LIN {X 0,Y 164.353,Z 359.01,A -85,B 0,C 180,E1 -23368.785,E2 -23368.785} C_VEL
LIN {X 0,Y 164.395,Z 359.001,A -85,B 0,C 180,E1 -23374.69,E2 -23374.69} C_VEL
LIN {X 0,Y 164.485,Z 358.995,A -85,B 0,C 180,E1 -23380.051,E2 -23380.051} C_VEL
LIN {X 0,Y 164.525,Z 358.989,A -85,B 0,C 180,E1 -23385.149,E2 -23385.149} C_VEL
LIN {X 0,Y 164.803,Z 358.955,A -85,B 0,C 180,E1 -23390.178,E2 -23390.178} C_VEL
LIN {X 0,Y 164.851,Z 358.949,A -85,B 0,C 180,E1 -23392.652,E2 -23392.652} C_VEL
LIN {X 0,Y 165.049,Z 358.926,A -85,B 0,C 180,E1 -23397.559,E2 -23397.559} C_VEL
LIN {X 0,Y 165.289,Z 358.897,A -85,B 0,C 180,E1 -23400,E2 -23400} C_VEL
LIN {X 0,Y 164.763,Z 358.963,A -85,B 0,C 180,E1 -23404.894,E2 -23404.894} C_VEL
LIN {X 0,Y 164.831,Z 358.955,A -85,B 0,C 180,E1 -23407.349,E2 -23407.349} C_VEL
LIN {X 0,Y 164.703,Z 358.969,A -85,B 0,C 180,E1 -23411.061,E2 -23411.061} C_VEL
LIN {X 0,Y 164.483,Z 358.999,A -85,B 0,C 180,E1 -23417.403,E2 -23417.403} C_VEL
LIN {X 0,Y 164.474,Z 358.998,A -85,B 0,C 180,E1 -23419.989,E2 -23419.989} C_VEL
LIN {X 0,Y 164.395,Z 359.008,A -85,B 0,C 180,E1 -23425.309,E2 -23425.309} C_VEL
LIN {X 0,Y 164.82,Z 361.559,A -85,B 0,C 180,E1 -23431.481,E2 -23431.481} C_VEL
LIN {X 0,Y 165.147,Z 364.035,A -85,B 0,C 180,E1 -23436.569,E2 -23436.569} C_VEL
LIN {X 0,Y 165.54,Z 366.68,A -85,B 0,C 180,E1 -23441.479,E2 -23441.479} C_VEL
LIN {X 0,Y 166.739,Z 369.834,A -85,B 0,C 180,E1 -23442.221,E2 -23442.221} C_VEL
LIN {X 0,Y 168.781,Z 372.777,A -85,B 0,C 180,E1 -23443.252,E2 -23443.252} C_VEL
LIN {X 0,Y 170.799,Z 376.689,A -85,B 0,C 180,E1 -23444.388,E2 -23444.388} C_VEL
LIN {X 0,Y 174.052,Z 383.605,A -85,B 0,C 180,E1 -23446.305,E2 -23446.305} C_VEL
LIN {X 0,Y 176.79,Z 390.925,A -85,B 0,C 180,E1 -23448.191,E2 -23448.191} C_VEL
LIN {X 0,Y 178.354,Z 398.431,A -85,B 0,C 180,E1 -23449.912,E2 -23449.912} C_VEL
LIN {X 0,Y 179.413,Z 408.097,A -85,B 0,C 180,E1 -23452.121,E2 -23452.121} C_VEL
LIN {X 0,Y 179.618,Z 418.57,A -85,B 0,C 180,E1 -23454.683,E2 -23454.683} C_VEL
LIN {X 0,Y 178.968,Z 428.265,A -85,B 0,C 180,E1 -23457.319,E2 -23457.319} C_VEL
LIN {X 0,Y 178.405,Z 432.364,A -85,B 0,C 180,E1 -23458.535,E2 -23458.535} C_VEL
LIN {X 0,Y 175.059,Z 441.2,A -85,B 0,C 180,E1 -23461.199,E2 -23461.199} C_VEL
LIN {X 0,Y 172.159,Z 448.374,A -85,B 0,C 180,E1 -23463.91,E2 -23463.91} C_VEL
LIN {X 0,Y 168.88,Z 455.682,A -85,B 0,C 180,E1 -23467.359,E2 -23467.359} C_VEL
LIN {X 0,Y 166.696,Z 460.537,A -85,B 0,C 180,E1 -23470.288,E2 -23470.288} C_VEL
LIN {X 0,Y 164.537,Z 465.256,A -85,B 0,C 180,E1 -23473.88,E2 -23473.88} C_VEL
LIN {X 0,Y 163.144,Z 468.87,A -85,B 0,C 180,E1 -23477.561,E2 -23477.561} C_VEL
LIN {X 0,Y 162.461,Z 470.733,A -85,B 0,C 180,E1 -23480.035,E2 -23480.035} C_VEL
LIN {X 0,Y 161.852,Z 473.135,A -85,B 0,C 180,E1 -23485.017,E2 -23485.017} C_VEL
LIN {X 0,Y 161.797,Z 473.748,A -85,B 0,C 180,E1 -23487.509,E2 -23487.509} C_VEL
LIN {X 0,Y 161.893,Z 473.964,A -85,B 0,C 180,E1 -23489.999,E2 -23489.999} C_VEL
LIN {X 0,Y 161.797,Z 473.737,A -85,B 0,C 180,E1 -23492.488,E2 -23492.488} C_VEL
LIN {X 0,Y 161.851,Z 473.118,A -85,B 0,C 180,E1 -23494.981,E2 -23494.981} C_VEL
LIN {X 0,Y 162.035,Z 472.109,A -85,B 0,C 180,E1 -23497.475,E2 -23497.475} C_VEL
LIN {X 0,Y 162.46,Z 470.698,A -85,B 0,C 180,E1 -23499.963,E2 -23499.963} C_VEL
LIN {X 0,Y 163.562,Z 467.743,A -85,B 0,C 180,E1 -23503.668,E2 -23503.668} C_VEL
LIN {X 0,Y 165.152,Z 463.748,A -85,B 0,C 180,E1 -23507.329,E2 -23507.329} C_VEL
LIN {X 0,Y 167.969,Z 457.619,A -85,B 0,C 180,E1 -23511.474,E2 -23511.474} C_VEL
LIN {X 0,Y 170.947,Z 451.054,A -85,B 0,C 180,E1 -23514.857,E2 -23514.857} C_VEL
LIN {X 0,Y 173.3,Z 445.244,A -85,B 0,C 180,E1 -23517.303,E2 -23517.303} C_VEL
LIN {X 0,Y 174.216,Z 441.463,A -85,B 0,C 180,E1 -23518.769,E2 -23518.769} C_VEL
LIN {X 0,Y 174.238,Z 437.625,A -85,B 0,C 180,E1 -23520.281,E2 -23520.281} C_VEL
LIN {X 0,Y 173.009,Z 426.964,A -85,B 0,C 180,E1 -23524.249,E2 -23524.249} C_VEL
LIN {X 0,Y 173.036,Z 423.996,A -85,B 0,C 180,E1 -23525.153,E2 -23525.153} C_VEL
LIN {X 0,Y 173.396,Z 414.41,A -85,B 0,C 180,E1 -23527.76,E2 -23527.76} C_VEL
LIN {X 0,Y 172.882,Z 404.098,A -85,B 0,C 180,E1 -23530.339,E2 -23530.339} C_VEL
LIN {X 0,Y 171.558,Z 395.307,A -85,B 0,C 180,E1 -23532.491,E2 -23532.491} C_VEL
LIN {X 0,Y 169.041,Z 387.542,A -85,B 0,C 180,E1 -23534.604,E2 -23534.604} C_VEL
LIN {X 0,Y 165.953,Z 380.904,A -85,B 0,C 180,E1 -23536.66,E2 -23536.66} C_VEL
LIN {X 0,Y 163.83,Z 376.649,A -85,B 0,C 180,E1 -23538.014,E2 -23538.014} C_VEL
LIN {X 0,Y 161.813,Z 372.888,A -85,B 0,C 180,E1 -23539.276,E2 -23539.276} C_VEL
LIN {X 0,Y 160.79,Z 371.257,A -85,B 0,C 180,E1 -23539.868,E2 -23539.868} C_VEL
LIN {X 0,Y 158.767,Z 367.896,A -85,B 0,C 180,E1 -23541.098,E2 -23541.098} C_VEL
LIN {X 0,Y 158.284,Z 366.287,A -85,B 0,C 180,E1 -23541.566,E2 -23541.566} C_VEL
LIN {X 0,Y 158.063,Z 364.741,A -85,B 0,C 180,E1 -23544.688,E2 -23544.688} C_VEL
LIN {X 0,Y 157.879,Z 363.325,A -85,B 0,C 180,E1 -23547.752,E2 -23547.752} C_VEL
LIN {X 0,Y 157.498,Z 360.965,A -85,B 0,C 180,E1 -23553.498,E2 -23553.498} C_VEL
LIN {X 0,Y 157.295,Z 359.957,A -85,B 0,C 180,E1 -23556.289,E2 -23556.289} C_VEL
LIN {X 0,Y 157.405,Z 359.877,A -85,B 0,C 180,E1 -23561.787,E2 -23561.787} C_VEL
LIN {X 0,Y 157.542,Z 359.86,A -85,B 0,C 180,E1 -23567.112,E2 -23567.112} C_VEL
LIN {X 0,Y 157.741,Z 359.835,A -85,B 0,C 180,E1 -23569.734,E2 -23569.734} C_VEL
LIN {X 0,Y 157.807,Z 359.828,A -85,B 0,C 180,E1 -23572.322,E2 -23572.322} C_VEL
LIN {X 0,Y 158.246,Z 359.771,A -85,B 0,C 180,E1 -23580,E2 -23580} C_VEL
LIN {X 0,Y 157.815,Z 359.825,A -85,B 0,C 180,E1 -23587.678,E2 -23587.678} C_VEL
LIN {X 0,Y 157.672,Z 359.842,A -85,B 0,C 180,E1 -23591.311,E2 -23591.311} C_VEL
LIN {X 0,Y 157.449,Z 359.874,A -85,B 0,C 180,E1 -23595.535,E2 -23595.535} C_VEL
LIN {X 0,Y 157.362,Z 359.884,A -85,B 0,C 180,E1 -23600.934,E2 -23600.934} C_VEL
LIN {X 0,Y 157.305,Z 359.889,A -85,B 0,C 180,E1 -23606.682,E2 -23606.682} C_VEL
LIN {X 0,Y 157.263,Z 359.896,A -85,B 0,C 180,E1 -23612.431,E2 -23612.431} C_VEL
LIN {X 0,Y 157.275,Z 360.116,A -85,B 0,C 180,E1 -23616.456,E2 -23616.456} C_VEL
LIN {X 0,Y 157.298,Z 360.711,A -85,B 0,C 180,E1 -23618.163,E2 -23618.163} C_VEL
LIN {X 0,Y 158.359,Z 363.418,A -85,B 0,C 180,E1 -23618.941,E2 -23618.941} C_VEL
LIN {X 0,Y 160.846,Z 366.551,A -85,B 0,C 180,E1 -23620.375,E2 -23620.375} C_VEL
LIN {X 0,Y 162.74,Z 370.024,A -85,B 0,C 180,E1 -23621.604,E2 -23621.604} C_VEL
LIN {X 0,Y 163.87,Z 371.847,A -85,B 0,C 180,E1 -23622.284,E2 -23622.284} C_VEL
LIN {X 0,Y 166.98,Z 377.77,A -85,B 0,C 180,E1 -23624.318,E2 -23624.318} C_VEL
LIN {X 0,Y 170.348,Z 385.376,A -85,B 0,C 180,E1 -23626.767,E2 -23626.767} C_VEL
LIN {X 0,Y 172.965,Z 393.791,A -85,B 0,C 180,E1 -23629.227,E2 -23629.227} C_VEL
LIN {X 0,Y 174.476,Z 402.79,A -85,B 0,C 180,E1 -23631.718,E2 -23631.718} C_VEL
LIN {X 0,Y 175.187,Z 412.008,A -85,B 0,C 180,E1 -23634.384,E2 -23634.384} C_VEL
LIN {X 0,Y 175.109,Z 418.891,A -85,B 0,C 180,E1 -23636.507,E2 -23636.507} C_VEL
LIN {X 0,Y 171.621,Z 428.426,A -85,B 0,C 180,E1 -23639.195,E2 -23639.195} C_VEL
LIN {X 0,Y 168.381,Z 436.318,A -85,B 0,C 180,E1 -23641.996,E2 -23641.996} C_VEL
LIN {X 0,Y 164.694,Z 443.99,A -85,B 0,C 180,E1 -23645.416,E2 -23645.416} C_VEL
LIN {X 0,Y 161.143,Z 451.035,A -85,B 0,C 180,E1 -23649.581,E2 -23649.581} C_VEL
LIN {X 0,Y 158.778,Z 455.72,A -85,B 0,C 180,E1 -23653.281,E2 -23653.281} C_VEL
LIN {X 0,Y 157.001,Z 459.302,A -85,B 0,C 180,E1 -23657.068,E2 -23657.068} C_VEL
LIN {X 0,Y 156.157,Z 461.149,A -85,B 0,C 180,E1 -23659.63,E2 -23659.63} C_VEL
LIN {X 0,Y 155.58,Z 462.534,A -85,B 0,C 180,E1 -23662.213,E2 -23662.213} C_VEL
LIN {X 0,Y 154.905,Z 464.126,A -85,B 0,C 180,E1 -23667.401,E2 -23667.401} C_VEL
LIN {X 0,Y 154.879,Z 464.35,A -85,B 0,C 180,E1 -23670.001,E2 -23670.001} C_VEL
LIN {X 0,Y 154.976,Z 463.919,A -85,B 0,C 180,E1 -23673.9,E2 -23673.9} C_VEL
LIN {X 0,Y 155.515,Z 462.602,A -85,B 0,C 180,E1 -23677.793,E2 -23677.793} C_VEL
LIN {X 0,Y 156.164,Z 461.244,A -85,B 0,C 180,E1 -23680.372,E2 -23680.372} C_VEL
LIN {X 0,Y 157.501,Z 458.377,A -85,B 0,C 180,E1 -23684.208,E2 -23684.208} C_VEL
LIN {X 0,Y 159.461,Z 454.485,A -85,B 0,C 180,E1 -23687.97,E2 -23687.97} C_VEL
LIN {X 0,Y 161.987,Z 449.463,A -85,B 0,C 180,E1 -23691.641,E2 -23691.641} C_VEL
LIN {X 0,Y 165.187,Z 443.13,A -85,B 0,C 180,E1 -23695.18,E2 -23695.18} C_VEL
LIN {X 0,Y 168.859,Z 435.21,A -85,B 0,C 180,E1 -23698.597,E2 -23698.597} C_VEL
LIN {X 0,Y 172.096,Z 427.315,A -85,B 0,C 180,E1 -23701.31,E2 -23701.31} C_VEL
LIN {X 0,Y 175.172,Z 419.412,A -85,B 0,C 180,E1 -23703.481,E2 -23703.481} C_VEL
LIN {X 0,Y 175.141,Z 409.831,A -85,B 0,C 180,E1 -23706.414,E2 -23706.414} C_VEL
LIN {X 0,Y 174.237,Z 400.686,A -85,B 0,C 180,E1 -23709.03,E2 -23709.03} C_VEL
LIN {X 0,Y 172.483,Z 391.797,A -85,B 0,C 180,E1 -23711.52,E2 -23711.52} C_VEL
LIN {X 0,Y 169.319,Z 382.614,A -85,B 0,C 180,E1 -23714.274,E2 -23714.274} C_VEL
LIN {X 0,Y 165.221,Z 374.414,A -85,B 0,C 180,E1 -23717.034,E2 -23717.034} C_VEL
LIN {X 0,Y 162.756,Z 370.019,A -85,B 0,C 180,E1 -23718.607,E2 -23718.607} C_VEL
LIN {X 0,Y 160.857,Z 366.588,A -85,B 0,C 180,E1 -23719.839,E2 -23719.839} C_VEL
LIN {X 0,Y 157.969,Z 362.664,A -85,B 0,C 180,E1 -23721.554,E2 -23721.554} C_VEL
LIN {X 0,Y 157.322,Z 360.713,A -85,B 0,C 180,E1 -23722.081,E2 -23722.081} C_VEL
LIN {X 0,Y 157.278,Z 359.894,A -85,B 0,C 180,E1 -23724.485,E2 -23724.485} C_VEL
LIN {X 0,Y 157.28,Z 359.889,A -85,B 0,C 180,E1 -23728.104,E2 -23728.104} C_VEL
LIN {X 0,Y 157.31,Z 359.889,A -85,B 0,C 180,E1 -23733.464,E2 -23733.464} C_VEL
LIN {X 0,Y 157.393,Z 359.879,A -85,B 0,C 180,E1 -23739.67,E2 -23739.67} C_VEL
LIN {X 0,Y 157.455,Z 359.872,A -85,B 0,C 180,E1 -23744.466,E2 -23744.466} C_VEL
LIN {X 0,Y 157.727,Z 359.838,A -85,B 0,C 180,E1 -23749.733,E2 -23749.733} C_VEL
LIN {X 0,Y 157.808,Z 359.828,A -85,B 0,C 180,E1 -23752.322,E2 -23752.322} C_VEL
LIN {X 0,Y 158.252,Z 359.774,A -85,B 0,C 180,E1 -23760,E2 -23760} C_VEL
LIN {X 0,Y 157.768,Z 359.836,A -85,B 0,C 180,E1 -23767.68,E2 -23767.68} C_VEL
LIN {X 0,Y 157.638,Z 359.85,A -85,B 0,C 180,E1 -23771.236,E2 -23771.236} C_VEL
LIN {X 0,Y 157.453,Z 359.874,A -85,B 0,C 180,E1 -23775.534,E2 -23775.534} C_VEL
LIN {X 0,Y 157.368,Z 359.884,A -85,B 0,C 180,E1 -23780.933,E2 -23780.933} C_VEL
LIN {X 0,Y 157.309,Z 360.019,A -85,B 0,C 180,E1 -23783.709,E2 -23783.709} C_VEL
LIN {X 0,Y 157.506,Z 361.155,A -85,B 0,C 180,E1 -23786.822,E2 -23786.822} C_VEL
LIN {X 0,Y 157.912,Z 363.396,A -85,B 0,C 180,E1 -23792.281,E2 -23792.281} C_VEL
LIN {X 0,Y 158.272,Z 366.115,A -85,B 0,C 180,E1 -23797.974,E2 -23797.974} C_VEL
LIN {X 0,Y 158.312,Z 366.364,A -85,B 0,C 180,E1 -23798.426,E2 -23798.426} C_VEL
LIN {X 0,Y 159.319,Z 369.145,A -85,B 0,C 180,E1 -23799.151,E2 -23799.151} C_VEL
LIN {X 0,Y 161.764,Z 372.735,A -85,B 0,C 180,E1 -23800.567,E2 -23800.567} C_VEL
LIN {X 0,Y 163.614,Z 376.302,A -85,B 0,C 180,E1 -23801.744,E2 -23801.744} C_VEL
LIN {X 0,Y 164.947,Z 378.808,A -85,B 0,C 180,E1 -23802.563,E2 -23802.563} C_VEL
LIN {X 0,Y 168.731,Z 386.833,A -85,B 0,C 180,E1 -23805.079,E2 -23805.079} C_VEL
LIN {X 0,Y 171.42,Z 394.551,A -85,B 0,C 180,E1 -23807.241,E2 -23807.241} C_VEL
LIN {X 0,Y 172.895,Z 403.402,A -85,B 0,C 180,E1 -23809.429,E2 -23809.429} C_VEL
LIN {X 0,Y 173.449,Z 413.342,A -85,B 0,C 180,E1 -23811.9,E2 -23811.9} C_VEL
LIN {X 0,Y 173.197,Z 423.113,A -85,B 0,C 180,E1 -23814.541,E2 -23814.541} C_VEL
LIN {X 0,Y 172.16,Z 432.143,A -85,B 0,C 180,E1 -23817.255,E2 -23817.255} C_VEL
LIN {X 0,Y 170.986,Z 435.894,A -85,B 0,C 180,E1 -23818.394,E2 -23818.394} C_VEL
LIN {X 0,Y 167.504,Z 444.057,A -85,B 0,C 180,E1 -23821.15,E2 -23821.15} C_VEL
LIN {X 0,Y 163.992,Z 452.076,A -85,B 0,C 180,E1 -23824.623,E2 -23824.623} C_VEL
LIN {X 0,Y 160.925,Z 458.501,A -85,B 0,C 180,E1 -23828.209,E2 -23828.209} C_VEL
LIN {X 0,Y 158.373,Z 463.605,A -85,B 0,C 180,E1 -23831.902,E2 -23831.902} C_VEL
LIN {X 0,Y 156.631,Z 467.579,A -85,B 0,C 180,E1 -23835.712,E2 -23835.712} C_VEL
LIN {X 0,Y 155.458,Z 470.518,A -85,B 0,C 180,E1 -23839.581,E2 -23839.581} C_VEL
LIN {X 0,Y 154.757,Z 472.92,A -85,B 0,C 180,E1 -23844.788,E2 -23844.788} C_VEL
LIN {X 0,Y 154.712,Z 473.627,A -85,B 0,C 180,E1 -23847.982,E2 -23847.982} C_VEL
LIN {X 0,Y 154.794,Z 473.749,A -85,B 0,C 180,E1 -23849.999,E2 -23849.999} C_VEL
LIN {X 0,Y 154.699,Z 473.521,A -85,B 0,C 180,E1 -23852.603,E2 -23852.603} C_VEL
LIN {X 0,Y 154.757,Z 472.901,A -85,B 0,C 180,E1 -23855.21,E2 -23855.21} C_VEL
LIN {X 0,Y 154.98,Z 471.892,A -85,B 0,C 180,E1 -23857.818,E2 -23857.818} C_VEL
LIN {X 0,Y 155.456,Z 470.481,A -85,B 0,C 180,E1 -23860.417,E2 -23860.417} C_VEL
LIN {X 0,Y 156.63,Z 467.525,A -85,B 0,C 180,E1 -23864.286,E2 -23864.286} C_VEL
LIN {X 0,Y 158.371,Z 463.531,A -85,B 0,C 180,E1 -23868.096,E2 -23868.096} C_VEL
LIN {X 0,Y 161.322,Z 457.4,A -85,B 0,C 180,E1 -23872.406,E2 -23872.406} C_VEL
LIN {X 0,Y 164.722,Z 450.298,A -85,B 0,C 180,E1 -23876.158,E2 -23876.158} C_VEL
LIN {X 0,Y 168.114,Z 442.409,A -85,B 0,C 180,E1 -23879.418,E2 -23879.418} C_VEL
LIN {X 0,Y 171.641,Z 433.901,A -85,B 0,C 180,E1 -23882.159,E2 -23882.159} C_VEL
LIN {X 0,Y 172.781,Z 426.73,A -85,B 0,C 180,E1 -23884.357,E2 -23884.357} C_VEL
LIN {X 0,Y 173.036,Z 423.996,A -85,B 0,C 180,E1 -23885.153,E2 -23885.153} C_VEL
LIN {X 0,Y 172.687,Z 419.729,A -85,B 0,C 180,E1 -23886.491,E2 -23886.491} C_VEL
LIN {X 0,Y 171.451,Z 415.728,A -85,B 0,C 180,E1 -23887.905,E2 -23887.905} C_VEL
LIN {X 0,Y 168.105,Z 407.951,A -85,B 0,C 180,E1 -23890.782,E2 -23890.782} C_VEL
LIN {X 0,Y 166.636,Z 402.115,A -85,B 0,C 180,E1 -23892.582,E2 -23892.582} C_VEL
LIN {X 0,Y 165.321,Z 395.581,A -85,B 0,C 180,E1 -23894.395,E2 -23894.395} C_VEL
LIN {X 0,Y 163.025,Z 389.258,A -85,B 0,C 180,E1 -23896.389,E2 -23896.389} C_VEL
LIN {X 0,Y 159.585,Z 381.699,A -85,B 0,C 180,E1 -23898.969,E2 -23898.969} C_VEL
LIN {X 0,Y 156.809,Z 376.441,A -85,B 0,C 180,E1 -23900.93,E2 -23900.93} C_VEL
LIN {X 0,Y 154.709,Z 372.434,A -85,B 0,C 180,E1 -23902.445,E2 -23902.445} C_VEL
LIN {X 0,Y 151.861,Z 368.339,A -85,B 0,C 180,E1 -23904.35,E2 -23904.35} C_VEL
LIN {X 0,Y 151.071,Z 365.975,A -85,B 0,C 180,E1 -23905.055,E2 -23905.055} C_VEL
LIN {X 0,Y 150.802,Z 364.217,A -85,B 0,C 180,E1 -23909.16,E2 -23909.16} C_VEL
LIN {X 0,Y 150.593,Z 362.925,A -85,B 0,C 180,E1 -23912.458,E2 -23912.458} C_VEL
LIN {X 0,Y 150.279,Z 361,A -85,B 0,C 180,E1 -23918.029,E2 -23918.029} C_VEL
LIN {X 0,Y 150.354,Z 360.757,A -85,B 0,C 180,E1 -23920.901,E2 -23920.901} C_VEL
LIN {X 0,Y 150.445,Z 360.744,A -85,B 0,C 180,E1 -23926.493,E2 -23926.493} C_VEL
LIN {X 0,Y 150.658,Z 360.716,A -85,B 0,C 180,E1 -23929.246,E2 -23929.246} C_VEL
LIN {X 0,Y 150.744,Z 360.706,A -85,B 0,C 180,E1 -23931.96,E2 -23931.96} C_VEL
LIN {X 0,Y 151.208,Z 360.648,A -85,B 0,C 180,E1 -23940,E2 -23940} C_VEL
LIN {X 0,Y 150.75,Z 360.704,A -85,B 0,C 180,E1 -23948.04,E2 -23948.04} C_VEL
LIN {X 0,Y 150.608,Z 360.722,A -85,B 0,C 180,E1 -23951.505,E2 -23951.505} C_VEL
LIN {X 0,Y 150.356,Z 360.755,A -85,B 0,C 180,E1 -23956.287,E2 -23956.287} C_VEL
LIN {X 0,Y 150.345,Z 360.758,A -85,B 0,C 180,E1 -23960.791,E2 -23960.791} C_VEL
LIN {X 0,Y 150.234,Z 360.771,A -85,B 0,C 180,E1 -23967.279,E2 -23967.279} C_VEL
LIN {X 0,Y 150.204,Z 360.774,A -85,B 0,C 180,E1 -23972.629,E2 -23972.629} C_VEL
LIN {X 0,Y 150.223,Z 361.059,A -85,B 0,C 180,E1 -23974.559,E2 -23974.559} C_VEL
LIN {X 0,Y 151.303,Z 363.715,A -85,B 0,C 180,E1 -23975.495,E2 -23975.495} C_VEL
LIN {X 0,Y 153.858,Z 366.979,A -85,B 0,C 180,E1 -23977.218,E2 -23977.218} C_VEL
LIN {X 0,Y 155.877,Z 370.541,A -85,B 0,C 180,E1 -23978.703,E2 -23978.703} C_VEL
LIN {X 0,Y 157.095,Z 372.257,A -85,B 0,C 180,E1 -23979.502,E2 -23979.502} C_VEL
LIN {X 0,Y 161.032,Z 379.67,A -85,B 0,C 180,E1 -23982.399,E2 -23982.399} C_VEL
LIN {X 0,Y 164.489,Z 387.463,A -85,B 0,C 180,E1 -23985.171,E2 -23985.171} C_VEL
LIN {X 0,Y 166.872,Z 395.066,A -85,B 0,C 180,E1 -23987.637,E2 -23987.637} C_VEL
LIN {X 0,Y 168.396,Z 403.904,A -85,B 0,C 180,E1 -23990.304,E2 -23990.304} C_VEL
LIN {X 0,Y 169.005,Z 413.397,A -85,B 0,C 180,E1 -23993.234,E2 -23993.234} C_VEL
LIN {X 0,Y 168.812,Z 420.176,A -85,B 0,C 180,E1 -23995.444,E2 -23995.444} C_VEL
LIN {X 0,Y 165.544,Z 428.694,A -85,B 0,C 180,E1 -23997.952,E2 -23997.952} C_VEL
LIN {X 0,Y 162.145,Z 436.536,A -85,B 0,C 180,E1 -24000.818,E2 -24000.818} C_VEL
LIN {X 0,Y 158.275,Z 444.207,A -85,B 0,C 180,E1 -24004.348,E2 -24004.348} C_VEL
LIN {X 0,Y 154.492,Z 451.252,A -85,B 0,C 180,E1 -24008.66,E2 -24008.66} C_VEL
LIN {X 0,Y 151.996,Z 455.937,A -85,B 0,C 180,E1 -24012.511,E2 -24012.511} C_VEL
LIN {X 0,Y 150.075,Z 459.519,A -85,B 0,C 180,E1 -24016.46,E2 -24016.46} C_VEL
LIN {X 0,Y 149.17,Z 461.366,A -85,B 0,C 180,E1 -24019.139,E2 -24019.139} C_VEL
LIN {X 0,Y 148.544,Z 462.75,A -85,B 0,C 180,E1 -24021.841,E2 -24021.841} C_VEL
LIN {X 0,Y 147.825,Z 464.341,A -85,B 0,C 180,E1 -24027.276,E2 -24027.276} C_VEL
LIN {X 0,Y 147.782,Z 464.566,A -85,B 0,C 180,E1 -24030.001,E2 -24030.001} C_VEL
LIN {X 0,Y 147.84,Z 464.264,A -85,B 0,C 180,E1 -24033.339,E2 -24033.339} C_VEL
LIN {X 0,Y 148.503,Z 462.817,A -85,B 0,C 180,E1 -24038.163,E2 -24038.163} C_VEL
LIN {X 0,Y 149.175,Z 461.46,A -85,B 0,C 180,E1 -24040.863,E2 -24040.863} C_VEL
LIN {X 0,Y 150.621,Z 458.592,A -85,B 0,C 180,E1 -24044.871,E2 -24044.871} C_VEL
LIN {X 0,Y 152.728,Z 454.699,A -85,B 0,C 180,E1 -24048.792,E2 -24048.792} C_VEL
LIN {X 0,Y 155.414,Z 449.676,A -85,B 0,C 180,E1 -24052.606,E2 -24052.606} C_VEL
LIN {X 0,Y 158.8,Z 443.343,A -85,B 0,C 180,E1 -24056.269,E2 -24056.269} C_VEL
LIN {X 0,Y 162.577,Z 435.6,A -85,B 0,C 180,E1 -24059.726,E2 -24059.726} C_VEL
LIN {X 0,Y 166.072,Z 427.528,A -85,B 0,C 180,E1 -24062.583,E2 -24062.583} C_VEL
LIN {X 0,Y 168.881,Z 420.689,A -85,B 0,C 180,E1 -24064.542,E2 -24064.542} C_VEL
LIN {X 0,Y 169.034,Z 412.607,A -85,B 0,C 180,E1 -24067.196,E2 -24067.196} C_VEL
LIN {X 0,Y 168.399,Z 403.632,A -85,B 0,C 180,E1 -24069.959,E2 -24069.959} C_VEL
LIN {X 0,Y 166.92,Z 395.095,A -85,B 0,C 180,E1 -24072.537,E2 -24072.537} C_VEL
LIN {X 0,Y 164.187,Z 386.637,A -85,B 0,C 180,E1 -24075.303,E2 -24075.303} C_VEL
LIN {X 0,Y 160.745,Z 379.247,A -85,B 0,C 180,E1 -24078.01,E2 -24078.01} C_VEL
LIN {X 0,Y 158.597,Z 375.113,A -85,B 0,C 180,E1 -24079.602,E2 -24079.602} C_VEL
LIN {X 0,Y 156.455,Z 371.161,A -85,B 0,C 180,E1 -24081.176,E2 -24081.176} C_VEL
LIN {X 0,Y 154.328,Z 368.029,A -85,B 0,C 180,E1 -24082.644,E2 -24082.644} C_VEL
LIN {X 0,Y 153.426,Z 366.28,A -85,B 0,C 180,E1 -24083.329,E2 -24083.329} C_VEL
LIN {X 0,Y 150.951,Z 363.166,A -85,B 0,C 180,E1 -24085.023,E2 -24085.023} C_VEL
LIN {X 0,Y 150.239,Z 361.055,A -85,B 0,C 180,E1 -24085.75,E2 -24085.75} C_VEL
LIN {X 0,Y 150.189,Z 360.775,A -85,B 0,C 180,E1 -24089.02,E2 -24089.02} C_VEL
LIN {X 0,Y 150.239,Z 360.77,A -85,B 0,C 180,E1 -24092.723,E2 -24092.723} C_VEL
LIN {X 0,Y 150.35,Z 360.758,A -85,B 0,C 180,E1 -24099.21,E2 -24099.21} C_VEL
LIN {X 0,Y 150.362,Z 360.756,A -85,B 0,C 180,E1 -24103.713,E2 -24103.713} C_VEL
LIN {X 0,Y 150.649,Z 360.72,A -85,B 0,C 180,E1 -24109.245,E2 -24109.245} C_VEL
LIN {X 0,Y 150.743,Z 360.709,A -85,B 0,C 180,E1 -24111.96,E2 -24111.96} C_VEL
LIN {X 0,Y 151.213,Z 360.65,A -85,B 0,C 180,E1 -24120,E2 -24120} C_VEL
LIN {X 0,Y 150.705,Z 360.714,A -85,B 0,C 180,E1 -24128.042,E2 -24128.042} C_VEL
LIN {X 0,Y 150.578,Z 360.729,A -85,B 0,C 180,E1 -24131.437,E2 -24131.437} C_VEL
LIN {X 0,Y 150.361,Z 360.757,A -85,B 0,C 180,E1 -24136.287,E2 -24136.287} C_VEL
LIN {X 0,Y 150.35,Z 360.758,A -85,B 0,C 180,E1 -24140.79,E2 -24140.79} C_VEL
LIN {X 0,Y 150.444,Z 362.01,A -85,B 0,C 180,E1 -24144.862,E2 -24144.862} C_VEL
LIN {X 0,Y 150.817,Z 364.276,A -85,B 0,C 180,E1 -24150.837,E2 -24150.837} C_VEL
LIN {X 0,Y 151.094,Z 366.091,A -85,B 0,C 180,E1 -24154.837,E2 -24154.837} C_VEL
LIN {X 0,Y 152.414,Z 369.346,A -85,B 0,C 180,E1 -24155.907,E2 -24155.907} C_VEL
LIN {X 0,Y 154.641,Z 372.269,A -85,B 0,C 180,E1 -24157.362,E2 -24157.362} C_VEL
LIN {X 0,Y 156.729,Z 376.34,A -85,B 0,C 180,E1 -24158.887,E2 -24158.887} C_VEL
LIN {X 0,Y 157.796,Z 378.138,A -85,B 0,C 180,E1 -24159.603,E2 -24159.603} C_VEL
LIN {X 0,Y 160.451,Z 383.481,A -85,B 0,C 180,E1 -24161.532,E2 -24161.532} C_VEL
LIN {X 0,Y 163.958,Z 391.593,A -85,B 0,C 180,E1 -24164.271,E2 -24164.271} C_VEL
LIN {X 0,Y 165.863,Z 397.492,A -85,B 0,C 180,E1 -24166.082,E2 -24166.082} C_VEL
LIN {X 0,Y 166.917,Z 404.124,A -85,B 0,C 180,E1 -24167.866,E2 -24167.866} C_VEL
LIN {X 0,Y 167.4,Z 413.267,A -85,B 0,C 180,E1 -24170.3,E2 -24170.3} C_VEL
LIN {X 0,Y 167.045,Z 423.035,A -85,B 0,C 180,E1 -24173.071,E2 -24173.071} C_VEL
LIN {X 0,Y 165.927,Z 431.92,A -85,B 0,C 180,E1 -24175.86,E2 -24175.86} C_VEL
LIN {X 0,Y 164.936,Z 435.68,A -85,B 0,C 180,E1 -24177.092,E2 -24177.092} C_VEL
LIN {X 0,Y 160.654,Z 445.332,A -85,B 0,C 180,E1 -24180.518,E2 -24180.518} C_VEL
LIN {X 0,Y 157.006,Z 453.018,A -85,B 0,C 180,E1 -24184.123,E2 -24184.123} C_VEL
LIN {X 0,Y 154.294,Z 458.285,A -85,B 0,C 180,E1 -24187.221,E2 -24187.221} C_VEL
LIN {X 0,Y 151.628,Z 463.391,A -85,B 0,C 180,E1 -24191.067,E2 -24191.067} C_VEL
LIN {X 0,Y 149.725,Z 467.363,A -85,B 0,C 180,E1 -24195.038,E2 -24195.038} C_VEL
LIN {X 0,Y 148.446,Z 470.302,A -85,B 0,C 180,E1 -24199.083,E2 -24199.083} C_VEL
LIN {X 0,Y 147.948,Z 471.702,A -85,B 0,C 180,E1 -24201.806,E2 -24201.806} C_VEL
LIN {X 0,Y 147.69,Z 472.705,A -85,B 0,C 180,E1 -24204.538,E2 -24204.538} C_VEL
LIN {X 0,Y 147.624,Z 473.464,A -85,B 0,C 180,E1 -24208.73,E2 -24208.73} C_VEL
LIN {X 0,Y 147.63,Z 473.455,A -85,B 0,C 180,E1 -24211.361,E2 -24211.361} C_VEL
LIN {X 0,Y 147.689,Z 472.686,A -85,B 0,C 180,E1 -24215.46,E2 -24215.46} C_VEL
LIN {X 0,Y 147.947,Z 471.676,A -85,B 0,C 180,E1 -24218.192,E2 -24218.192} C_VEL
LIN {X 0,Y 148.445,Z 470.264,A -85,B 0,C 180,E1 -24220.915,E2 -24220.915} C_VEL
LIN {X 0,Y 149.723,Z 467.308,A -85,B 0,C 180,E1 -24224.96,E2 -24224.96} C_VEL
LIN {X 0,Y 151.627,Z 463.314,A -85,B 0,C 180,E1 -24228.931,E2 -24228.931} C_VEL
LIN {X 0,Y 154.742,Z 457.182,A -85,B 0,C 180,E1 -24233.414,E2 -24233.414} C_VEL
LIN {X 0,Y 158.068,Z 450.661,A -85,B 0,C 180,E1 -24237.013,E2 -24237.013} C_VEL
LIN {X 0,Y 161.946,Z 442.19,A -85,B 0,C 180,E1 -24240.656,E2 -24240.656} C_VEL
LIN {X 0,Y 165.53,Z 433.677,A -85,B 0,C 180,E1 -24243.499,E2 -24243.499} C_VEL
LIN {X 0,Y 166.738,Z 425.413,A -85,B 0,C 180,E1 -24246.162,E2 -24246.162} C_VEL
LIN {X 0,Y 167.324,Z 415.429,A -85,B 0,C 180,E1 -24249.05,E2 -24249.05} C_VEL
LIN {X 0,Y 167.005,Z 405.626,A -85,B 0,C 180,E1 -24251.672,E2 -24251.672} C_VEL
LIN {X 0,Y 166.636,Z 402.115,A -85,B 0,C 180,E1 -24252.582,E2 -24252.582} C_VEL
LIN {X 0,Y 165.893,Z 399.25,A -85,B 0,C 180,E1 -24253.464,E2 -24253.464} C_VEL
LIN {X 0,Y 163.76,Z 395.725,A -85,B 0,C 180,E1 -24254.942,E2 -24254.942} C_VEL
LIN {X 0,Y 156.201,Z 388.028,A -85,B 0,C 180,E1 -24259.28,E2 -24259.28} C_VEL
LIN {X 0,Y 154.066,Z 384.34,A -85,B 0,C 180,E1 -24260.883,E2 -24260.883} C_VEL
LIN {X 0,Y 152.711,Z 381.525,A -85,B 0,C 180,E1 -24261.999,E2 -24261.999} C_VEL
LIN {X 0,Y 150.359,Z 376.921,A -85,B 0,C 180,E1 -24263.939,E2 -24263.939} C_VEL
LIN {X 0,Y 148.205,Z 373.329,A -85,B 0,C 180,E1 -24265.66,E2 -24265.66} C_VEL
LIN {X 0,Y 147.444,Z 371.645,A -85,B 0,C 180,E1 -24266.339,E2 -24266.339} C_VEL
LIN {X 0,Y 144.848,Z 368.385,A -85,B 0,C 180,E1 -24268.357,E2 -24268.357} C_VEL
LIN {X 0,Y 143.853,Z 365.596,A -85,B 0,C 180,E1 -24269.442,E2 -24269.442} C_VEL
LIN {X 0,Y 143.561,Z 363.966,A -85,B 0,C 180,E1 -24273.858,E2 -24273.858} C_VEL
LIN {X 0,Y 143.352,Z 362.051,A -85,B 0,C 180,E1 -24279.929,E2 -24279.929} C_VEL
LIN {X 0,Y 143.299,Z 361.635,A -85,B 0,C 180,E1 -24282.887,E2 -24282.887} C_VEL
LIN {X 0,Y 143.589,Z 361.597,A -85,B 0,C 180,E1 -24288.71,E2 -24288.71} C_VEL
LIN {X 0,Y 143.664,Z 361.588,A -85,B 0,C 180,E1 -24291.561,E2 -24291.561} C_VEL
LIN {X 0,Y 144.167,Z 361.525,A -85,B 0,C 180,E1 -24300,E2 -24300} C_VEL
LIN {X 0,Y 143.669,Z 361.585,A -85,B 0,C 180,E1 -24308.439,E2 -24308.439} C_VEL
LIN {X 0,Y 143.543,Z 361.602,A -85,B 0,C 180,E1 -24311.713,E2 -24311.713} C_VEL
LIN {X 0,Y 143.296,Z 361.633,A -85,B 0,C 180,E1 -24317.114,E2 -24317.114} C_VEL
LIN {X 0,Y 143.27,Z 361.639,A -85,B 0,C 180,E1 -24321.253,E2 -24321.253} C_VEL
LIN {X 0,Y 143.178,Z 361.651,A -85,B 0,C 180,E1 -24327.932,E2 -24327.932} C_VEL
LIN {X 0,Y 143.107,Z 361.661,A -85,B 0,C 180,E1 -24330.224,E2 -24330.224} C_VEL
LIN {X 0,Y 143.943,Z 364.126,A -85,B 0,C 180,E1 -24331.148,E2 -24331.148} C_VEL
LIN {X 0,Y 145.947,Z 366.468,A -85,B 0,C 180,E1 -24332.776,E2 -24332.776} C_VEL
LIN {X 0,Y 147.079,Z 367.488,A -85,B 0,C 180,E1 -24333.607,E2 -24333.607} C_VEL
LIN {X 0,Y 149.221,Z 371.22,A -85,B 0,C 180,E1 -24335.443,E2 -24335.443} C_VEL
LIN {X 0,Y 150.235,Z 372.538,A -85,B 0,C 180,E1 -24336.2,E2 -24336.2} C_VEL
LIN {X 0,Y 155.092,Z 381.405,A -85,B 0,C 180,E1 -24340.222,E2 -24340.222} C_VEL
LIN {X 0,Y 158.566,Z 389.463,A -85,B 0,C 180,E1 -24343.393,E2 -24343.393} C_VEL
LIN {X 0,Y 160.968,Z 396.902,A -85,B 0,C 180,E1 -24346.086,E2 -24346.086} C_VEL
LIN {X 0,Y 162.259,Z 404.071,A -85,B 0,C 180,E1 -24348.456,E2 -24348.456} C_VEL
LIN {X 0,Y 162.865,Z 413.118,A -85,B 0,C 180,E1 -24351.425,E2 -24351.425} C_VEL
LIN {X 0,Y 162.598,Z 421.449,A -85,B 0,C 180,E1 -24354.304,E2 -24354.304} C_VEL
LIN {X 0,Y 158.452,Z 431.32,A -85,B 0,C 180,E1 -24357.43,E2 -24357.43} C_VEL
LIN {X 0,Y 154.558,Z 439.484,A -85,B 0,C 180,E1 -24360.739,E2 -24360.739} C_VEL
LIN {X 0,Y 150.662,Z 446.645,A -85,B 0,C 180,E1 -24364.44,E2 -24364.44} C_VEL
LIN {X 0,Y 147.887,Z 451.47,A -85,B 0,C 180,E1 -24367.657,E2 -24367.657} C_VEL
LIN {X 0,Y 145.249,Z 456.153,A -85,B 0,C 180,E1 -24371.671,E2 -24371.671} C_VEL
LIN {X 0,Y 143.18,Z 459.735,A -85,B 0,C 180,E1 -24375.795,E2 -24375.795} C_VEL
LIN {X 0,Y 142.208,Z 461.582,A -85,B 0,C 180,E1 -24378.6,E2 -24378.6} C_VEL
LIN {X 0,Y 141.514,Z 462.966,A -85,B 0,C 180,E1 -24381.433,E2 -24381.433} C_VEL
LIN {X 0,Y 141.016,Z 463.952,A -85,B 0,C 180,E1 -24384.281,E2 -24384.281} C_VEL
LIN {X 0,Y 140.69,Z 464.781,A -85,B 0,C 180,E1 -24390.001,E2 -24390.001} C_VEL
LIN {X 0,Y 140.737,Z 464.585,A -85,B 0,C 180,E1 -24392.864,E2 -24392.864} C_VEL
LIN {X 0,Y 141.009,Z 463.999,A -85,B 0,C 180,E1 -24395.722,E2 -24395.722} C_VEL
LIN {X 0,Y 142.212,Z 461.674,A -85,B 0,C 180,E1 -24401.402,E2 -24401.402} C_VEL
LIN {X 0,Y 143.771,Z 458.807,A -85,B 0,C 180,E1 -24405.597,E2 -24405.597} C_VEL
LIN {X 0,Y 146.034,Z 454.913,A -85,B 0,C 180,E1 -24409.688,E2 -24409.688} C_VEL
LIN {X 0,Y 148.894,Z 449.89,A -85,B 0,C 180,E1 -24413.655,E2 -24413.655} C_VEL
LIN {X 0,Y 152.478,Z 443.556,A -85,B 0,C 180,E1 -24417.447,E2 -24417.447} C_VEL
LIN {X 0,Y 156.336,Z 436.046,A -85,B 0,C 180,E1 -24420.922,E2 -24420.922} C_VEL
LIN {X 0,Y 160.208,Z 427.565,A -85,B 0,C 180,E1 -24424.008,E2 -24424.008} C_VEL
LIN {X 0,Y 162.629,Z 421.919,A -85,B 0,C 180,E1 -24425.691,E2 -24425.691} C_VEL
LIN {X 0,Y 162.938,Z 412.136,A -85,B 0,C 180,E1 -24429.068,E2 -24429.068} C_VEL
LIN {X 0,Y 162.248,Z 403.752,A -85,B 0,C 180,E1 -24431.84,E2 -24431.84} C_VEL
LIN {X 0,Y 161.139,Z 397.231,A -85,B 0,C 180,E1 -24433.977,E2 -24433.977} C_VEL
LIN {X 0,Y 158.675,Z 389.687,A -85,B 0,C 180,E1 -24436.728,E2 -24436.728} C_VEL
LIN {X 0,Y 155.271,Z 381.895,A -85,B 0,C 180,E1 -24439.834,E2 -24439.834} C_VEL
LIN {X 0,Y 152.393,Z 376.379,A -85,B 0,C 180,E1 -24442.25,E2 -24442.25} C_VEL
LIN {X 0,Y 150.286,Z 372.575,A -85,B 0,C 180,E1 -24444.022,E2 -24444.022} C_VEL
LIN {X 0,Y 147.378,Z 368.183,A -85,B 0,C 180,E1 -24446.374,E2 -24446.374} C_VEL
LIN {X 0,Y 146.705,Z 367.035,A -85,B 0,C 180,E1 -24446.957,E2 -24446.957} C_VEL
LIN {X 0,Y 144.281,Z 364.705,A -85,B 0,C 180,E1 -24448.832,E2 -24448.832} C_VEL
LIN {X 0,Y 143.231,Z 362.316,A -85,B 0,C 180,E1 -24449.906,E2 -24449.906} C_VEL
LIN {X 0,Y 143.111,Z 361.655,A -85,B 0,C 180,E1 -24450.183,E2 -24450.183} C_VEL
LIN {X 0,Y 143.151,Z 361.65,A -85,B 0,C 180,E1 -24453.777,E2 -24453.777} C_VEL
LIN {X 0,Y 143.307,Z 361.633,A -85,B 0,C 180,E1 -24459.922,E2 -24459.922} C_VEL
LIN {X 0,Y 143.365,Z 361.625,A -85,B 0,C 180,E1 -24465.812,E2 -24465.812} C_VEL
LIN {X 0,Y 143.596,Z 361.597,A -85,B 0,C 180,E1 -24468.71,E2 -24468.71} C_VEL
LIN {X 0,Y 143.662,Z 361.59,A -85,B 0,C 180,E1 -24471.561,E2 -24471.561} C_VEL
LIN {X 0,Y 144.172,Z 361.527,A -85,B 0,C 180,E1 -24480,E2 -24480} C_VEL
LIN {X 0,Y 143.626,Z 361.595,A -85,B 0,C 180,E1 -24488.441,E2 -24488.441} C_VEL
LIN {X 0,Y 143.506,Z 361.611,A -85,B 0,C 180,E1 -24491.629,E2 -24491.629} C_VEL
LIN {X 0,Y 143.301,Z 361.638,A -85,B 0,C 180,E1 -24497.113,E2 -24497.113} C_VEL
LIN {X 0,Y 143.409,Z 362.497,A -85,B 0,C 180,E1 -24501.388,E2 -24501.388} C_VEL
LIN {X 0,Y 143.568,Z 364.03,A -85,B 0,C 180,E1 -24506.14,E2 -24506.14} C_VEL
LIN {X 0,Y 143.862,Z 365.721,A -85,B 0,C 180,E1 -24510.454,E2 -24510.454} C_VEL
LIN {X 0,Y 145.105,Z 368.815,A -85,B 0,C 180,E1 -24511.682,E2 -24511.682} C_VEL
LIN {X 0,Y 147.774,Z 372.119,A -85,B 0,C 180,E1 -24513.745,E2 -24513.745} C_VEL
LIN {X 0,Y 149.587,Z 375.904,A -85,B 0,C 180,E1 -24515.343,E2 -24515.343} C_VEL
LIN {X 0,Y 151.089,Z 378.195,A -85,B 0,C 180,E1 -24516.479,E2 -24516.479} C_VEL
LIN {X 0,Y 154.03,Z 384.224,A -85,B 0,C 180,E1 -24518.942,E2 -24518.942} C_VEL
LIN {X 0,Y 156.148,Z 388.794,A -85,B 0,C 180,E1 -24520.74,E2 -24520.74} C_VEL
LIN {X 0,Y 159.098,Z 396.258,A -85,B 0,C 180,E1 -24523.47,E2 -24523.47} C_VEL
LIN {X 0,Y 160.605,Z 401.949,A -85,B 0,C 180,E1 -24525.324,E2 -24525.324} C_VEL
LIN {X 0,Y 161.352,Z 409.383,A -85,B 0,C 180,E1 -24527.47,E2 -24527.47} C_VEL
LIN {X 0,Y 161.292,Z 418.142,A -85,B 0,C 180,E1 -24530.007,E2 -24530.007} C_VEL
LIN {X 0,Y 160.489,Z 427.594,A -85,B 0,C 180,E1 -24532.977,E2 -24532.977} C_VEL
LIN {X 0,Y 158.941,Z 435.465,A -85,B 0,C 180,E1 -24535.682,E2 -24535.682} C_VEL
LIN {X 0,Y 154.487,Z 445.118,A -85,B 0,C 180,E1 -24539.216,E2 -24539.216} C_VEL
LIN {X 0,Y 150.606,Z 452.803,A -85,B 0,C 180,E1 -24542.936,E2 -24542.936} C_VEL
LIN {X 0,Y 147.711,Z 458.069,A -85,B 0,C 180,E1 -24546.144,E2 -24546.144} C_VEL
LIN {X 0,Y 144.919,Z 463.176,A -85,B 0,C 180,E1 -24550.154,E2 -24550.154} C_VEL
LIN {X 0,Y 142.847,Z 467.147,A -85,B 0,C 180,E1 -24554.299,E2 -24554.299} C_VEL
LIN {X 0,Y 141.455,Z 470.086,A -85,B 0,C 180,E1 -24558.536,E2 -24558.536} C_VEL
LIN {X 0,Y 140.621,Z 472.489,A -85,B 0,C 180,E1 -24564.262,E2 -24564.262} C_VEL
LIN {X 0,Y 140.569,Z 473.29,A -85,B 0,C 180,E1 -24569.355,E2 -24569.355} C_VEL
LIN {X 0,Y 140.508,Z 473.089,A -85,B 0,C 180,E1 -24572.866,E2 -24572.866} C_VEL
LIN {X 0,Y 140.621,Z 472.47,A -85,B 0,C 180,E1 -24575.735,E2 -24575.735} C_VEL
LIN {X 0,Y 141.453,Z 470.047,A -85,B 0,C 180,E1 -24581.462,E2 -24581.462} C_VEL
LIN {X 0,Y 142.845,Z 467.09,A -85,B 0,C 180,E1 -24585.698,E2 -24585.698} C_VEL
LIN {X 0,Y 144.917,Z 463.097,A -85,B 0,C 180,E1 -24589.843,E2 -24589.843} C_VEL
LIN {X 0,Y 148.23,Z 456.964,A -85,B 0,C 180,E1 -24594.509,E2 -24594.509} C_VEL
LIN {X 0,Y 151.218,Z 451.512,A -85,B 0,C 180,E1 -24597.693,E2 -24597.693} C_VEL
LIN {X 0,Y 155.119,Z 443.463,A -85,B 0,C 180,E1 -24601.4,E2 -24601.4} C_VEL
LIN {X 0,Y 158.904,Z 435.266,A -85,B 0,C 180,E1 -24604.324,E2 -24604.324} C_VEL
LIN {X 0,Y 160.41,Z 427.349,A -85,B 0,C 180,E1 -24607.042,E2 -24607.042} C_VEL
LIN {X 0,Y 161.242,Z 417.845,A -85,B 0,C 180,E1 -24610.005,E2 -24610.005} C_VEL
LIN {X 0,Y 161.164,Z 407.16,A -85,B 0,C 180,E1 -24613.078,E2 -24613.078} C_VEL
LIN {X 0,Y 160.38,Z 400.937,A -85,B 0,C 180,E1 -24614.895,E2 -24614.895} C_VEL
LIN {X 0,Y 158.476,Z 394.496,A -85,B 0,C 180,E1 -24617.038,E2 -24617.038} C_VEL
LIN {X 0,Y 155.325,Z 386.826,A -85,B 0,C 180,E1 -24619.852,E2 -24619.852} C_VEL
LIN {X 0,Y 154.066,Z 384.34,A -85,B 0,C 180,E1 -24620.883,E2 -24620.883} C_VEL
LIN {X 0,Y 152.107,Z 380.741,A -85,B 0,C 180,E1 -24622.468,E2 -24622.468} C_VEL
LIN {X 0,Y 149.622,Z 377.96,A -85,B 0,C 180,E1 -24624.217,E2 -24624.217} C_VEL
LIN {X 0,Y 144.041,Z 373.912,A -85,B 0,C 180,E1 -24628.073,E2 -24628.073} C_VEL
LIN {X 0,Y 140.49,Z 371.459,A -85,B 0,C 180,E1 -24630.832,E2 -24630.832} C_VEL
LIN {X 0,Y 137.829,Z 368.308,A -85,B 0,C 180,E1 -24633.4,E2 -24633.4} C_VEL
LIN {X 0,Y 136.538,Z 365.135,A -85,B 0,C 180,E1 -24635.075,E2 -24635.075} C_VEL
LIN {X 0,Y 136.457,Z 363.99,A -85,B 0,C 180,E1 -24638.868,E2 -24638.868} C_VEL
LIN {X 0,Y 136.27,Z 362.51,A -85,B 0,C 180,E1 -24645.056,E2 -24645.056} C_VEL
LIN {X 0,Y 136.492,Z 362.483,A -85,B 0,C 180,E1 -24648.114,E2 -24648.114} C_VEL
LIN {X 0,Y 136.59,Z 362.469,A -85,B 0,C 180,E1 -24651.12,E2 -24651.12} C_VEL
LIN {X 0,Y 137.125,Z 362.402,A -85,B 0,C 180,E1 -24660,E2 -24660} C_VEL
LIN {X 0,Y 136.594,Z 362.467,A -85,B 0,C 180,E1 -24668.88,E2 -24668.88} C_VEL
LIN {X 0,Y 136.487,Z 362.482,A -85,B 0,C 180,E1 -24671.955,E2 -24671.955} C_VEL
LIN {X 0,Y 136.236,Z 362.515,A -85,B 0,C 180,E1 -24678.031,E2 -24678.031} C_VEL
LIN {X 0,Y 136.191,Z 362.519,A -85,B 0,C 180,E1 -24681.746,E2 -24681.746} C_VEL
LIN {X 0,Y 136.062,Z 362.535,A -85,B 0,C 180,E1 -24684.713,E2 -24684.713} C_VEL
LIN {X 0,Y 136.786,Z 364.789,A -85,B 0,C 180,E1 -24685.793,E2 -24685.793} C_VEL
LIN {X 0,Y 138.376,Z 366.892,A -85,B 0,C 180,E1 -24687.515,E2 -24687.515} C_VEL
LIN {X 0,Y 140.257,Z 368.303,A -85,B 0,C 180,E1 -24689.222,E2 -24689.222} C_VEL
LIN {X 0,Y 141.905,Z 371.488,A -85,B 0,C 180,E1 -24691.023,E2 -24691.023} C_VEL
LIN {X 0,Y 143.945,Z 373.747,A -85,B 0,C 180,E1 -24692.796,E2 -24692.796} C_VEL
LIN {X 0,Y 146.176,Z 377.536,A -85,B 0,C 180,E1 -24694.921,E2 -24694.921} C_VEL
LIN {X 0,Y 150.2,Z 385.502,A -85,B 0,C 180,E1 -24698.834,E2 -24698.834} C_VEL
LIN {X 0,Y 153.018,Z 392.12,A -85,B 0,C 180,E1 -24701.758,E2 -24701.758} C_VEL
LIN {X 0,Y 155.226,Z 399.19,A -85,B 0,C 180,E1 -24704.568,E2 -24704.568} C_VEL
LIN {X 0,Y 156.346,Z 405.647,A -85,B 0,C 180,E1 -24706.926,E2 -24706.926} C_VEL
LIN {X 0,Y 156.796,Z 414.28,A -85,B 0,C 180,E1 -24709.969,E2 -24709.969} C_VEL
LIN {X 0,Y 156.473,Z 421.684,A -85,B 0,C 180,E1 -24712.676,E2 -24712.676} C_VEL
LIN {X 0,Y 156.125,Z 423.615,A -85,B 0,C 180,E1 -24713.386,E2 -24713.386} C_VEL
LIN {X 0,Y 152.07,Z 432.431,A -85,B 0,C 180,E1 -24716.32,E2 -24716.32} C_VEL
LIN {X 0,Y 148.411,Z 439.702,A -85,B 0,C 180,E1 -24719.401,E2 -24719.401} C_VEL
LIN {X 0,Y 144.3,Z 446.862,A -85,B 0,C 180,E1 -24723.225,E2 -24723.225} C_VEL
LIN {X 0,Y 141.334,Z 451.687,A -85,B 0,C 180,E1 -24726.561,E2 -24726.561} C_VEL
LIN {X 0,Y 138.519,Z 456.37,A -85,B 0,C 180,E1 -24730.746,E2 -24730.746} C_VEL
LIN {X 0,Y 136.315,Z 459.951,A -85,B 0,C 180,E1 -24735.063,E2 -24735.063} C_VEL
LIN {X 0,Y 135.249,Z 461.798,A -85,B 0,C 180,E1 -24738.005,E2 -24738.005} C_VEL
LIN {X 0,Y 134.487,Z 463.182,A -85,B 0,C 180,E1 -24740.982,E2 -24740.982} C_VEL
LIN {X 0,Y 133.956,Z 464.168,A -85,B 0,C 180,E1 -24743.978,E2 -24743.978} C_VEL
LIN {X 0,Y 133.596,Z 464.907,A -85,B 0,C 180,E1 -24748.238,E2 -24748.238} C_VEL
LIN {X 0,Y 133.66,Z 464.8,A -85,B 0,C 180,E1 -24753.015,E2 -24753.015} C_VEL
LIN {X 0,Y 133.952,Z 464.214,A -85,B 0,C 180,E1 -24756.025,E2 -24756.025} C_VEL
LIN {X 0,Y 135.252,Z 461.889,A -85,B 0,C 180,E1 -24761.997,E2 -24761.997} C_VEL
LIN {X 0,Y 136.955,Z 459.021,A -85,B 0,C 180,E1 -24766.395,E2 -24766.395} C_VEL
LIN {X 0,Y 139.357,Z 455.128,A -85,B 0,C 180,E1 -24770.673,E2 -24770.673} C_VEL
LIN {X 0,Y 142.403,Z 450.104,A -85,B 0,C 180,E1 -24774.804,E2 -24774.804} C_VEL
LIN {X 0,Y 146.228,Z 443.768,A -85,B 0,C 180,E1 -24778.727,E2 -24778.727} C_VEL
LIN {X 0,Y 150.142,Z 436.535,A -85,B 0,C 180,E1 -24782.2,E2 -24782.2} C_VEL
LIN {X 0,Y 154.375,Z 427.775,A -85,B 0,C 180,E1 -24785.483,E2 -24785.483} C_VEL
LIN {X 0,Y 156.057,Z 424.074,A -85,B 0,C 180,E1 -24786.635,E2 -24786.635} C_VEL
LIN {X 0,Y 156.684,Z 420.091,A -85,B 0,C 180,E1 -24788.08,E2 -24788.08} C_VEL
LIN {X 0,Y 156.822,Z 411.652,A -85,B 0,C 180,E1 -24791.148,E2 -24791.148} C_VEL
LIN {X 0,Y 156.014,Z 402.594,A -85,B 0,C 180,E1 -24794.346,E2 -24794.346} C_VEL
LIN {X 0,Y 154.352,Z 395.826,A -85,B 0,C 180,E1 -24796.922,E2 -24796.922} C_VEL
LIN {X 0,Y 151.514,Z 388.426,A -85,B 0,C 180,E1 -24800.092,E2 -24800.092} C_VEL
LIN {X 0,Y 148.624,Z 382.056,A -85,B 0,C 180,E1 -24803.006,E2 -24803.006} C_VEL
LIN {X 0,Y 145.86,Z 377.085,A -85,B 0,C 180,E1 -24805.622,E2 -24805.622} C_VEL
LIN {X 0,Y 143.405,Z 372.931,A -85,B 0,C 180,E1 -24808.001,E2 -24808.001} C_VEL
LIN {X 0,Y 141.226,Z 370.471,A -85,B 0,C 180,E1 -24809.95,E2 -24809.95} C_VEL
LIN {X 0,Y 139.97,Z 367.991,A -85,B 0,C 180,E1 -24811.37,E2 -24811.37} C_VEL
LIN {X 0,Y 137.408,Z 365.828,A -85,B 0,C 180,E1 -24813.823,E2 -24813.823} C_VEL
LIN {X 0,Y 136.298,Z 363.617,A -85,B 0,C 180,E1 -24815.231,E2 -24815.231} C_VEL
LIN {X 0,Y 136.075,Z 362.528,A -85,B 0,C 180,E1 -24815.689,E2 -24815.689} C_VEL
LIN {X 0,Y 136.242,Z 362.514,A -85,B 0,C 180,E1 -24818.832,E2 -24818.832} C_VEL
LIN {X 0,Y 136.273,Z 362.508,A -85,B 0,C 180,E1 -24825.056,E2 -24825.056} C_VEL
LIN {X 0,Y 136.499,Z 362.48,A -85,B 0,C 180,E1 -24828.115,E2 -24828.115} C_VEL
LIN {X 0,Y 136.59,Z 362.469,A -85,B 0,C 180,E1 -24831.12,E2 -24831.12} C_VEL
LIN {X 0,Y 137.13,Z 362.405,A -85,B 0,C 180,E1 -24840,E2 -24840} C_VEL
LIN {X 0,Y 136.552,Z 362.476,A -85,B 0,C 180,E1 -24848.882,E2 -24848.882} C_VEL
LIN {X 0,Y 136.442,Z 362.492,A -85,B 0,C 180,E1 -24851.89,E2 -24851.89} C_VEL
LIN {X 0,Y 136.268,Z 362.528,A -85,B 0,C 180,E1 -24854.944,E2 -24854.944} C_VEL
LIN {X 0,Y 136.485,Z 364.051,A -85,B 0,C 180,E1 -24861.128,E2 -24861.128} C_VEL
LIN {X 0,Y 136.547,Z 365.154,A -85,B 0,C 180,E1 -24864.72,E2 -24864.72} C_VEL
LIN {X 0,Y 137.63,Z 367.956,A -85,B 0,C 180,E1 -24866.131,E2 -24866.131} C_VEL
LIN {X 0,Y 140.04,Z 371.03,A -85,B 0,C 180,E1 -24868.556,E2 -24868.556} C_VEL
LIN {X 0,Y 140.962,Z 372.089,A -85,B 0,C 180,E1 -24869.401,E2 -24869.401} C_VEL
LIN {X 0,Y 142.598,Z 375.539,A -85,B 0,C 180,E1 -24871.165,E2 -24871.165} C_VEL
LIN {X 0,Y 144.335,Z 377.938,A -85,B 0,C 180,E1 -24872.696,E2 -24872.696} C_VEL
LIN {X 0,Y 146.322,Z 382.02,A -85,B 0,C 180,E1 -24874.671,E2 -24874.671} C_VEL
LIN {X 0,Y 147.386,Z 384.058,A -85,B 0,C 180,E1 -24875.658,E2 -24875.658} C_VEL
LIN {X 0,Y 151.161,Z 392.455,A -85,B 0,C 180,E1 -24879.372,E2 -24879.372} C_VEL
LIN {X 0,Y 153.874,Z 400.026,A -85,B 0,C 180,E1 -24882.352,E2 -24882.352} C_VEL
LIN {X 0,Y 155.261,Z 406.271,A -85,B 0,C 180,E1 -24884.555,E2 -24884.555} C_VEL
LIN {X 0,Y 155.524,Z 415.272,A -85,B 0,C 180,E1 -24887.325,E2 -24887.325} C_VEL
LIN {X 0,Y 154.776,Z 425.197,A -85,B 0,C 180,E1 -24890.527,E2 -24890.527} C_VEL
LIN {X 0,Y 153.422,Z 433.437,A -85,B 0,C 180,E1 -24893.451,E2 -24893.451} C_VEL
LIN {X 0,Y 152.316,Z 437.041,A -85,B 0,C 180,E1 -24894.776,E2 -24894.776} C_VEL
LIN {X 0,Y 148.389,Z 444.904,A -85,B 0,C 180,E1 -24897.803,E2 -24897.803} C_VEL
LIN {X 0,Y 144.275,Z 452.587,A -85,B 0,C 180,E1 -24901.643,E2 -24901.643} C_VEL
LIN {X 0,Y 140.173,Z 459.677,A -85,B 0,C 180,E1 -24906.352,E2 -24906.352} C_VEL
LIN {X 0,Y 137.379,Z 464.395,A -85,B 0,C 180,E1 -24910.577,E2 -24910.577} C_VEL
LIN {X 0,Y 135.418,Z 468.007,A -85,B 0,C 180,E1 -24914.959,E2 -24914.959} C_VEL
LIN {X 0,Y 134.487,Z 469.871,A -85,B 0,C 180,E1 -24917.933,E2 -24917.933} C_VEL
LIN {X 0,Y 133.547,Z 472.274,A -85,B 0,C 180,E1 -24923.957,E2 -24923.957} C_VEL
LIN {X 0,Y 133.412,Z 472.886,A -85,B 0,C 180,E1 -24926.979,E2 -24926.979} C_VEL
LIN {X 0,Y 133.532,Z 473.104,A -85,B 0,C 180,E1 -24929.999,E2 -24929.999} C_VEL
LIN {X 0,Y 133.411,Z 472.874,A -85,B 0,C 180,E1 -24933.018,E2 -24933.018} C_VEL
LIN {X 0,Y 133.547,Z 472.254,A -85,B 0,C 180,E1 -24936.04,E2 -24936.04} C_VEL
LIN {X 0,Y 134.486,Z 469.83,A -85,B 0,C 180,E1 -24942.064,E2 -24942.064} C_VEL
LIN {X 0,Y 135.974,Z 466.872,A -85,B 0,C 180,E1 -24946.514,E2 -24946.514} C_VEL
LIN {X 0,Y 138.222,Z 462.879,A -85,B 0,C 180,E1 -24950.848,E2 -24950.848} C_VEL
LIN {X 0,Y 141.787,Z 456.746,A -85,B 0,C 180,E1 -24955.702,E2 -24955.702} C_VEL
LIN {X 0,Y 145.399,Z 450.303,A -85,B 0,C 180,E1 -24959.536,E2 -24959.536} C_VEL
LIN {X 0,Y 149.858,Z 441.753,A -85,B 0,C 180,E1 -24963.437,E2 -24963.437} C_VEL
LIN {X 0,Y 152.914,Z 435.041,A -85,B 0,C 180,E1 -24965.871,E2 -24965.871} C_VEL
LIN {X 0,Y 154.613,Z 425.985,A -85,B 0,C 180,E1 -24969.117,E2 -24969.117} C_VEL
LIN {X 0,Y 155.338,Z 417.6,A -85,B 0,C 180,E1 -24971.859,E2 -24971.859} C_VEL
LIN {X 0,Y 155.387,Z 408.777,A -85,B 0,C 180,E1 -24974.574,E2 -24974.574} C_VEL
LIN {X 0,Y 154.761,Z 403.516,A -85,B 0,C 180,E1 -24976.26,E2 -24976.26} C_VEL
LIN {X 0,Y 153.187,Z 397.983,A -85,B 0,C 180,E1 -24978.299,E2 -24978.299} C_VEL
LIN {X 0,Y 149.683,Z 389.104,A -85,B 0,C 180,E1 -24981.939,E2 -24981.939} C_VEL
LIN {X 0,Y 146.168,Z 381.819,A -85,B 0,C 180,E1 -24985.287,E2 -24985.287} C_VEL
LIN {X 0,Y 143.719,Z 377.022,A -85,B 0,C 180,E1 -24987.666,E2 -24987.666} C_VEL
LIN {X 0,Y 141.442,Z 373.491,A -85,B 0,C 180,E1 -24989.795,E2 -24989.795} C_VEL
LIN {X 0,Y 140.81,Z 371.693,A -85,B 0,C 180,E1 -24990.565,E2 -24990.565} C_VEL
LIN {X 0,Y 140.49,Z 371.459,A -85,B 0,C 180,E1 -24990.832,E2 -24990.832} C_VEL
LIN {X 0,Y 138.165,Z 370.458,A -85,B 0,C 180,E1 -24992.753,E2 -24992.753} C_VEL
LIN {X 0,Y 133.065,Z 370.118,A -85,B 0,C 180,E1 -24997.375,E2 -24997.375} C_VEL
LIN {X 0,Y 131.738,Z 369.288,A -85,B 0,C 180,E1 -24998.966,E2 -24998.966} C_VEL
LIN {X 0,Y 129.945,Z 366.257,A -85,B 0,C 180,E1 -25001.881,E2 -25001.881} C_VEL
LIN {X 0,Y 129.374,Z 364.563,A -85,B 0,C 180,E1 -25003.226,E2 -25003.226} C_VEL
LIN {X 0,Y 129.433,Z 363.59,A -85,B 0,C 180,E1 -25007.775,E2 -25007.775} C_VEL
LIN {X 0,Y 129.515,Z 363.352,A -85,B 0,C 180,E1 -25010.631,E2 -25010.631} C_VEL
LIN {X 0,Y 130.081,Z 363.279,A -85,B 0,C 180,E1 -25020,E2 -25020} C_VEL
LIN {X 0,Y 129.518,Z 363.35,A -85,B 0,C 180,E1 -25029.369,E2 -25029.369} C_VEL
LIN {X 0,Y 129.388,Z 363.368,A -85,B 0,C 180,E1 -25032.549,E2 -25032.549} C_VEL
LIN {X 0,Y 129.181,Z 363.527,A -85,B 0,C 180,E1 -25037.003,E2 -25037.003} C_VEL
LIN {X 0,Y 130.16,Z 366.215,A -85,B 0,C 180,E1 -25039.108,E2 -25039.108} C_VEL
LIN {X 0,Y 132.646,Z 368.716,A -85,B 0,C 180,E1 -25042.622,E2 -25042.622} C_VEL
LIN {X 0,Y 133.581,Z 369.375,A -85,B 0,C 180,E1 -25043.754,E2 -25043.754} C_VEL
LIN {X 0,Y 135.162,Z 372.549,A -85,B 0,C 180,E1 -25046.023,E2 -25046.023} C_VEL
LIN {X 0,Y 137.33,Z 374.678,A -85,B 0,C 180,E1 -25048.358,E2 -25048.358} C_VEL
LIN {X 0,Y 138.987,Z 377.783,A -85,B 0,C 180,E1 -25050.375,E2 -25050.375} C_VEL
LIN {X 0,Y 140.284,Z 379.136,A -85,B 0,C 180,E1 -25051.61,E2 -25051.61} C_VEL
LIN {X 0,Y 144.324,Z 387.168,A -85,B 0,C 180,E1 -25056.201,E2 -25056.201} C_VEL
LIN {X 0,Y 147.626,Z 395.215,A -85,B 0,C 180,E1 -25060.171,E2 -25060.171} C_VEL
LIN {X 0,Y 149.541,Z 401.591,A -85,B 0,C 180,E1 -25062.998,E2 -25062.998} C_VEL
LIN {X 0,Y 150.612,Z 408.061,A -85,B 0,C 180,E1 -25065.58,E2 -25065.58} C_VEL
LIN {X 0,Y 150.809,Z 416.358,A -85,B 0,C 180,E1 -25068.742,E2 -25068.742} C_VEL
LIN {X 0,Y 150.22,Z 423.844,A -85,B 0,C 180,E1 -25071.694,E2 -25071.694} C_VEL
LIN {X 0,Y 148.746,Z 427.574,A -85,B 0,C 180,E1 -25072.959,E2 -25072.959} C_VEL
LIN {X 0,Y 144.247,Z 436.447,A -85,B 0,C 180,E1 -25076.341,E2 -25076.341} C_VEL
LIN {X 0,Y 140.109,Z 443.695,A -85,B 0,C 180,E1 -25079.896,E2 -25079.896} C_VEL
LIN {X 0,Y 136.063,Z 450.099,A -85,B 0,C 180,E1 -25083.959,E2 -25083.959} C_VEL
LIN {X 0,Y 132.798,Z 455.172,A -85,B 0,C 180,E1 -25088.258,E2 -25088.258} C_VEL
LIN {X 0,Y 130.178,Z 459.11,A -85,B 0,C 180,E1 -25092.728,E2 -25092.728} C_VEL
LIN {X 0,Y 128.301,Z 462.015,A -85,B 0,C 180,E1 -25097.345,E2 -25097.345} C_VEL
LIN {X 0,Y 127.489,Z 463.398,A -85,B 0,C 180,E1 -25100.482,E2 -25100.482} C_VEL
LIN {X 0,Y 126.585,Z 464.987,A -85,B 0,C 180,E1 -25106.819,E2 -25106.819} C_VEL
LIN {X 0,Y 126.505,Z 465.212,A -85,B 0,C 180,E1 -25110.001,E2 -25110.001} C_VEL
LIN {X 0,Y 126.585,Z 465.015,A -85,B 0,C 180,E1 -25113.184,E2 -25113.184} C_VEL
LIN {X 0,Y 127.477,Z 463.461,A -85,B 0,C 180,E1 -25119.521,E2 -25119.521} C_VEL
LIN {X 0,Y 128.303,Z 462.104,A -85,B 0,C 180,E1 -25122.658,E2 -25122.658} C_VEL
LIN {X 0,Y 130.141,Z 459.236,A -85,B 0,C 180,E1 -25127.28,E2 -25127.28} C_VEL
LIN {X 0,Y 132.731,Z 455.342,A -85,B 0,C 180,E1 -25131.756,E2 -25131.756} C_VEL
LIN {X 0,Y 135.981,Z 450.318,A -85,B 0,C 180,E1 -25136.061,E2 -25136.061} C_VEL
LIN {X 0,Y 140.042,Z 443.982,A -85,B 0,C 180,E1 -25140.123,E2 -25140.123} C_VEL
LIN {X 0,Y 144.845,Z 435.518,A -85,B 0,C 180,E1 -25144.226,E2 -25144.226} C_VEL
LIN {X 0,Y 149.543,Z 426.21,A -85,B 0,C 180,E1 -25147.659,E2 -25147.659} C_VEL
LIN {X 0,Y 150.247,Z 424.293,A -85,B 0,C 180,E1 -25148.301,E2 -25148.301} C_VEL
LIN {X 0,Y 150.907,Z 416.863,A -85,B 0,C 180,E1 -25151.238,E2 -25151.238} C_VEL
LIN {X 0,Y 150.664,Z 407.954,A -85,B 0,C 180,E1 -25154.653,E2 -25154.653} C_VEL
LIN {X 0,Y 149.761,Z 402.264,A -85,B 0,C 180,E1 -25156.922,E2 -25156.922} C_VEL
LIN {X 0,Y 147.397,Z 394.457,A -85,B 0,C 180,E1 -25160.413,E2 -25160.413} C_VEL
LIN {X 0,Y 144.208,Z 386.869,A -85,B 0,C 180,E1 -25164.209,E2 -25164.209} C_VEL
LIN {X 0,Y 141.754,Z 382.077,A -85,B 0,C 180,E1 -25166.95,E2 -25166.95} C_VEL
LIN {X 0,Y 140.067,Z 378.934,A -85,B 0,C 180,E1 -25168.891,E2 -25168.891} C_VEL
LIN {X 0,Y 137.794,Z 375.756,A -85,B 0,C 180,E1 -25171.33,E2 -25171.33} C_VEL
LIN {X 0,Y 137.047,Z 374.277,A -85,B 0,C 180,E1 -25172.306,E2 -25172.306} C_VEL
LIN {X 0,Y 134.703,Z 371.871,A -85,B 0,C 180,E1 -25174.918,E2 -25174.918} C_VEL
LIN {X 0,Y 133.531,Z 369.135,A -85,B 0,C 180,E1 -25176.75,E2 -25176.75} C_VEL
LIN {X 0,Y 130.642,Z 366.942,A -85,B 0,C 180,E1 -25180.557,E2 -25180.557} C_VEL
LIN {X 0,Y 129.329,Z 364.182,A -85,B 0,C 180,E1 -25183.118,E2 -25183.118} C_VEL
LIN {X 0,Y 129.171,Z 363.395,A -85,B 0,C 180,E1 -25183.606,E2 -25183.606} C_VEL
LIN {X 0,Y 129.418,Z 363.362,A -85,B 0,C 180,E1 -25187.82,E2 -25187.82} C_VEL
LIN {X 0,Y 129.516,Z 363.349,A -85,B 0,C 180,E1 -25190.631,E2 -25190.631} C_VEL
LIN {X 0,Y 130.086,Z 363.282,A -85,B 0,C 180,E1 -25200,E2 -25200} C_VEL
LIN {X 0,Y 129.475,Z 363.358,A -85,B 0,C 180,E1 -25209.372,E2 -25209.372} C_VEL
LIN {X 0,Y 129.383,Z 363.74,A -85,B 0,C 180,E1 -25212.549,E2 -25212.549} C_VEL
LIN {X 0,Y 129.399,Z 364.641,A -85,B 0,C 180,E1 -25216.567,E2 -25216.567} C_VEL
LIN {X 0,Y 130.758,Z 367.94,A -85,B 0,C 180,E1 -25219.221,E2 -25219.221} C_VEL
LIN {X 0,Y 134.08,Z 371.798,A -85,B 0,C 180,E1 -25223.696,E2 -25223.696} C_VEL
LIN {X 0,Y 136.01,Z 375.799,A -85,B 0,C 180,E1 -25226.363,E2 -25226.363} C_VEL
LIN {X 0,Y 137.837,Z 378.146,A -85,B 0,C 180,E1 -25228.348,E2 -25228.348} C_VEL
LIN {X 0,Y 139.836,Z 382.171,A -85,B 0,C 180,E1 -25230.733,E2 -25230.733} C_VEL
LIN {X 0,Y 141.069,Z 384.558,A -85,B 0,C 180,E1 -25232.12,E2 -25232.12} C_VEL
LIN {X 0,Y 143.684,Z 390.19,A -85,B 0,C 180,E1 -25235.08,E2 -25235.08} C_VEL
LIN {X 0,Y 146.61,Z 397.54,A -85,B 0,C 180,E1 -25238.548,E2 -25238.548} C_VEL
LIN {X 0,Y 149.075,Z 405.632,A -85,B 0,C 180,E1 -25241.969,E2 -25241.969} C_VEL
LIN {X 0,Y 149.797,Z 410.442,A -85,B 0,C 180,E1 -25243.75,E2 -25243.75} C_VEL
LIN {X 0,Y 149.536,Z 419.318,A -85,B 0,C 180,E1 -25246.695,E2 -25246.695} C_VEL
LIN {X 0,Y 148.414,Z 428.206,A -85,B 0,C 180,E1 -25249.812,E2 -25249.812} C_VEL
LIN {X 0,Y 147.029,Z 435.024,A -85,B 0,C 180,E1 -25252.45,E2 -25252.45} C_VEL
LIN {X 0,Y 145.711,Z 438.498,A -85,B 0,C 180,E1 -25253.782,E2 -25253.782} C_VEL
LIN {X 0,Y 140.814,Z 447.561,A -85,B 0,C 180,E1 -25257.636,E2 -25257.636} C_VEL
LIN {X 0,Y 136.756,Z 454.612,A -85,B 0,C 180,E1 -25261.616,E2 -25261.616} C_VEL
LIN {X 0,Y 133.65,Z 459.462,A -85,B 0,C 180,E1 -25265.122,E2 -25265.122} C_VEL
LIN {X 0,Y 130.672,Z 464.18,A -85,B 0,C 180,E1 -25269.537,E2 -25269.537} C_VEL
LIN {X 0,Y 128.551,Z 467.792,A -85,B 0,C 180,E1 -25274.135,E2 -25274.135} C_VEL
LIN {X 0,Y 127.516,Z 469.655,A -85,B 0,C 180,E1 -25277.263,E2 -25277.263} C_VEL
LIN {X 0,Y 126.469,Z 472.058,A -85,B 0,C 180,E1 -25283.618,E2 -25283.618} C_VEL
LIN {X 0,Y 126.315,Z 472.671,A -85,B 0,C 180,E1 -25286.809,E2 -25286.809} C_VEL
LIN {X 0,Y 126.445,Z 472.889,A -85,B 0,C 180,E1 -25289.999,E2 -25289.999} C_VEL
LIN {X 0,Y 126.314,Z 472.658,A -85,B 0,C 180,E1 -25293.188,E2 -25293.188} C_VEL
LIN {X 0,Y 126.468,Z 472.037,A -85,B 0,C 180,E1 -25296.38,E2 -25296.38} C_VEL
LIN {X 0,Y 127.514,Z 469.613,A -85,B 0,C 180,E1 -25302.734,E2 -25302.734} C_VEL
LIN {X 0,Y 129.144,Z 466.655,A -85,B 0,C 180,E1 -25307.414,E2 -25307.414} C_VEL
LIN {X 0,Y 131.582,Z 462.661,A -85,B 0,C 180,E1 -25311.953,E2 -25311.953} C_VEL
LIN {X 0,Y 135.419,Z 456.529,A -85,B 0,C 180,E1 -25317.006,E2 -25317.006} C_VEL
LIN {X 0,Y 138.874,Z 450.709,A -85,B 0,C 180,E1 -25320.647,E2 -25320.647} C_VEL
LIN {X 0,Y 143.134,Z 443.025,A -85,B 0,C 180,E1 -25324.376,E2 -25324.376} C_VEL
LIN {X 0,Y 146.414,Z 436.613,A -85,B 0,C 180,E1 -25326.868,E2 -25326.868} C_VEL
LIN {X 0,Y 148.01,Z 429.983,A -85,B 0,C 180,E1 -25329.442,E2 -25329.442} C_VEL
LIN {X 0,Y 149.256,Z 421.394,A -85,B 0,C 180,E1 -25332.507,E2 -25332.507} C_VEL
LIN {X 0,Y 149.734,Z 411.558,A -85,B 0,C 180,E1 -25335.783,E2 -25335.783} C_VEL
LIN {X 0,Y 149.281,Z 406.749,A -85,B 0,C 180,E1 -25337.472,E2 -25337.472} C_VEL
LIN {X 0,Y 147.734,Z 400.873,A -85,B 0,C 180,E1 -25339.864,E2 -25339.864} C_VEL
LIN {X 0,Y 144.867,Z 393.007,A -85,B 0,C 180,E1 -25343.391,E2 -25343.391} C_VEL
LIN {X 0,Y 142.331,Z 387.273,A -85,B 0,C 180,E1 -25346.255,E2 -25346.255} C_VEL
LIN {X 0,Y 139.815,Z 382.184,A -85,B 0,C 180,E1 -25349.078,E2 -25349.078} C_VEL
LIN {X 0,Y 137.874,Z 378.362,A -85,B 0,C 180,E1 -25351.349,E2 -25351.349} C_VEL
LIN {X 0,Y 137.199,Z 377.216,A -85,B 0,C 180,E1 -25352.133,E2 -25352.133} C_VEL
LIN {X 0,Y 134.841,Z 373.831,A -85,B 0,C 180,E1 -25354.843,E2 -25354.843} C_VEL
LIN {X 0,Y 133.841,Z 371.381,A -85,B 0,C 180,E1 -25356.345,E2 -25356.345} C_VEL
LIN {X 0,Y 131.738,Z 369.288,A -85,B 0,C 180,E1 -25358.966,E2 -25358.966} C_VEL
LIN {X 0,Y 129.959,Z 368.063,A -85,B 0,C 180,E1 -25361.384,E2 -25361.384} C_VEL
LIN {X 0,Y 127.1,Z 367.922,A -85,B 0,C 180,E1 -25365.633,E2 -25365.633} C_VEL
LIN {X 0,Y 124.518,Z 368.241,A -85,B 0,C 180,E1 -25371.007,E2 -25371.007} C_VEL
LIN {X 0,Y 124.006,Z 367.855,A -85,B 0,C 180,E1 -25372.834,E2 -25372.834} C_VEL
LIN {X 0,Y 123.365,Z 365.652,A -85,B 0,C 180,E1 -25380,E2 -25380} C_VEL
LIN {X 0,Y 127.188,Z 370.344,A -85,B 0,C 180,E1 -25396.142,E2 -25396.142} C_VEL
LIN {X 0,Y 128.273,Z 373.185,A -85,B 0,C 180,E1 -25398.777,E2 -25398.777} C_VEL
LIN {X 0,Y 131.004,Z 376.007,A -85,B 0,C 180,E1 -25402.993,E2 -25402.993} C_VEL
LIN {X 0,Y 132.312,Z 378.705,A -85,B 0,C 180,E1 -25405.147,E2 -25405.147} C_VEL
LIN {X 0,Y 133.443,Z 380.001,A -85,B 0,C 180,E1 -25406.593,E2 -25406.593} C_VEL
LIN {X 0,Y 136.832,Z 385.216,A -85,B 0,C 180,E1 -25410.906,E2 -25410.906} C_VEL
LIN {X 0,Y 140.029,Z 392.32,A -85,B 0,C 180,E1 -25415.253,E2 -25415.253} C_VEL
LIN {X 0,Y 142.579,Z 399.203,A -85,B 0,C 180,E1 -25418.937,E2 -25418.937} C_VEL
LIN {X 0,Y 144.357,Z 406.25,A -85,B 0,C 180,E1 -25422.324,E2 -25422.324} C_VEL
LIN {X 0,Y 144.967,Z 411.671,A -85,B 0,C 180,E1 -25424.663,E2 -25424.663} C_VEL
LIN {X 0,Y 144.767,Z 420.072,A -85,B 0,C 180,E1 -25428.127,E2 -25428.127} C_VEL
LIN {X 0,Y 143.952,Z 425.998,A -85,B 0,C 180,E1 -25430.606,E2 -25430.606} C_VEL
LIN {X 0,Y 139.052,Z 435.442,A -85,B 0,C 180,E1 -25434.167,E2 -25434.167} C_VEL
LIN {X 0,Y 134.014,Z 443.913,A -85,B 0,C 180,E1 -25438.373,E2 -25438.373} C_VEL
LIN {X 0,Y 129.713,Z 450.316,A -85,B 0,C 180,E1 -25442.58,E2 -25442.58} C_VEL
LIN {X 0,Y 126.224,Z 455.389,A -85,B 0,C 180,E1 -25447.063,E2 -25447.063} C_VEL
LIN {X 0,Y 123.403,Z 459.327,A -85,B 0,C 180,E1 -25451.748,E2 -25451.748} C_VEL
LIN {X 0,Y 121.384,Z 462.231,A -85,B 0,C 180,E1 -25456.611,E2 -25456.611} C_VEL
LIN {X 0,Y 120.487,Z 463.614,A -85,B 0,C 180,E1 -25459.924,E2 -25459.924} C_VEL
LIN {X 0,Y 119.498,Z 465.203,A -85,B 0,C 180,E1 -25466.63,E2 -25466.63} C_VEL
LIN {X 0,Y 119.419,Z 465.427,A -85,B 0,C 180,E1 -25470.001,E2 -25470.001} C_VEL
LIN {X 0,Y 119.499,Z 465.23,A -85,B 0,C 180,E1 -25473.373,E2 -25473.373} C_VEL
LIN {X 0,Y 120.479,Z 463.676,A -85,B 0,C 180,E1 -25480.08,E2 -25480.08} C_VEL
LIN {X 0,Y 121.385,Z 462.319,A -85,B 0,C 180,E1 -25483.392,E2 -25483.392} C_VEL
LIN {X 0,Y 123.363,Z 459.451,A -85,B 0,C 180,E1 -25488.261,E2 -25488.261} C_VEL
LIN {X 0,Y 126.162,Z 455.556,A -85,B 0,C 180,E1 -25492.952,E2 -25492.952} C_VEL
LIN {X 0,Y 129.637,Z 450.532,A -85,B 0,C 180,E1 -25497.44,E2 -25497.44} C_VEL
LIN {X 0,Y 133.94,Z 444.195,A -85,B 0,C 180,E1 -25501.65,E2 -25501.65} C_VEL
LIN {X 0,Y 138.746,Z 436.227,A -85,B 0,C 180,E1 -25505.657,E2 -25505.657} C_VEL
LIN {X 0,Y 143.936,Z 426.424,A -85,B 0,C 180,E1 -25509.402,E2 -25509.402} C_VEL
LIN {X 0,Y 144.8,Z 421.091,A -85,B 0,C 180,E1 -25511.625,E2 -25511.625} C_VEL
LIN {X 0,Y 145.078,Z 413.378,A -85,B 0,C 180,E1 -25514.849,E2 -25514.849} C_VEL
LIN {X 0,Y 144.703,Z 407.867,A -85,B 0,C 180,E1 -25517.159,E2 -25517.159} C_VEL
LIN {X 0,Y 143.174,Z 401.067,A -85,B 0,C 180,E1 -25520.347,E2 -25520.347} C_VEL
LIN {X 0,Y 140.224,Z 392.643,A -85,B 0,C 180,E1 -25524.803,E2 -25524.803} C_VEL
LIN {X 0,Y 137.008,Z 385.65,A -85,B 0,C 180,E1 -25529.138,E2 -25529.138} C_VEL
LIN {X 0,Y 134.724,Z 382.086,A -85,B 0,C 180,E1 -25531.998,E2 -25531.998} C_VEL
LIN {X 0,Y 134.133,Z 380.601,A -85,B 0,C 180,E1 -25532.966,E2 -25532.966} C_VEL
LIN {X 0,Y 131.734,Z 377.727,A -85,B 0,C 180,E1 -25536.101,E2 -25536.101} C_VEL
LIN {X 0,Y 130.719,Z 375.525,A -85,B 0,C 180,E1 -25537.892,E2 -25537.892} C_VEL
LIN {X 0,Y 128.125,Z 372.903,A -85,B 0,C 180,E1 -25542.028,E2 -25542.028} C_VEL
LIN {X 0,Y 127.047,Z 370.123,A -85,B 0,C 180,E1 -25544.766,E2 -25544.766} C_VEL
LIN {X 0,Y 123.581,Z 366.148,A -85,B 0,C 180,E1 -25560,E2 -25560} C_VEL
LIN {X 0,Y 125.784,Z 369.762,A -85,B 0,C 180,E1 -25572.018,E2 -25572.018} C_VEL
LIN {X 0,Y 127.479,Z 371.46,A -85,B 0,C 180,E1 -25575.693,E2 -25575.693} C_VEL
LIN {X 0,Y 129.005,Z 375.053,A -85,B 0,C 180,E1 -25579.079,E2 -25579.079} C_VEL
LIN {X 0,Y 131.387,Z 378.106,A -85,B 0,C 180,E1 -25582.714,E2 -25582.714} C_VEL
LIN {X 0,Y 132.781,Z 381.411,A -85,B 0,C 180,E1 -25585.052,E2 -25585.052} C_VEL
LIN {X 0,Y 134.6,Z 384.179,A -85,B 0,C 180,E1 -25587.421,E2 -25587.421} C_VEL
LIN {X 0,Y 135.972,Z 387.355,A -85,B 0,C 180,E1 -25589.408,E2 -25589.408} C_VEL
LIN {X 0,Y 137.076,Z 389.561,A -85,B 0,C 180,E1 -25590.844,E2 -25590.844} C_VEL
LIN {X 0,Y 140.231,Z 397.374,A -85,B 0,C 180,E1 -25595.194,E2 -25595.194} C_VEL
LIN {X 0,Y 143.106,Z 406.633,A -85,B 0,C 180,E1 -25599.675,E2 -25599.675} C_VEL
LIN {X 0,Y 144.076,Z 411.944,A -85,B 0,C 180,E1 -25601.952,E2 -25601.952} C_VEL
LIN {X 0,Y 143.932,Z 418.505,A -85,B 0,C 180,E1 -25604.335,E2 -25604.335} C_VEL
LIN {X 0,Y 142.773,Z 427.344,A -85,B 0,C 180,E1 -25607.593,E2 -25607.593} C_VEL
LIN {X 0,Y 141.141,Z 434.799,A -85,B 0,C 180,E1 -25610.589,E2 -25610.589} C_VEL
LIN {X 0,Y 139.977,Z 438.283,A -85,B 0,C 180,E1 -25612.044,E2 -25612.044} C_VEL
LIN {X 0,Y 134.922,Z 447.211,A -85,B 0,C 180,E1 -25615.946,E2 -25615.946} C_VEL
LIN {X 0,Y 130.777,Z 453.948,A -85,B 0,C 180,E1 -25619.831,E2 -25619.831} C_VEL
LIN {X 0,Y 127.201,Z 459.246,A -85,B 0,C 180,E1 -25623.767,E2 -25623.767} C_VEL
LIN {X 0,Y 124.019,Z 463.965,A -85,B 0,C 180,E1 -25628.385,E2 -25628.385} C_VEL
LIN {X 0,Y 121.699,Z 467.576,A -85,B 0,C 180,E1 -25633.216,E2 -25633.216} C_VEL
LIN {X 0,Y 120.575,Z 469.439,A -85,B 0,C 180,E1 -25636.516,E2 -25636.516} C_VEL
LIN {X 0,Y 119.415,Z 471.843,A -85,B 0,C 180,E1 -25643.239,E2 -25643.239} C_VEL
LIN {X 0,Y 119.229,Z 472.455,A -85,B 0,C 180,E1 -25646.619,E2 -25646.619} C_VEL
LIN {X 0,Y 119.36,Z 472.674,A -85,B 0,C 180,E1 -25649.999,E2 -25649.999} C_VEL
LIN {X 0,Y 119.414,Z 471.821,A -85,B 0,C 180,E1 -25656.758,E2 -25656.758} C_VEL
LIN {X 0,Y 120.574,Z 469.396,A -85,B 0,C 180,E1 -25663.481,E2 -25663.481} C_VEL
LIN {X 0,Y 122.358,Z 466.437,A -85,B 0,C 180,E1 -25668.414,E2 -25668.414} C_VEL
LIN {X 0,Y 125.001,Z 462.444,A -85,B 0,C 180,E1 -25673.174,E2 -25673.174} C_VEL
LIN {X 0,Y 129.132,Z 456.312,A -85,B 0,C 180,E1 -25678.436,E2 -25678.436} C_VEL
LIN {X 0,Y 133.325,Z 449.616,A -85,B 0,C 180,E1 -25682.703,E2 -25682.703} C_VEL
LIN {X 0,Y 138.188,Z 441.315,A -85,B 0,C 180,E1 -25686.695,E2 -25686.695} C_VEL
LIN {X 0,Y 140.589,Z 436.387,A -85,B 0,C 180,E1 -25688.67,E2 -25688.67} C_VEL
LIN {X 0,Y 142.383,Z 429.022,A -85,B 0,C 180,E1 -25691.678,E2 -25691.678} C_VEL
LIN {X 0,Y 143.61,Z 420.73,A -85,B 0,C 180,E1 -25694.782,E2 -25694.782} C_VEL
LIN {X 0,Y 144.088,Z 413.034,A -85,B 0,C 180,E1 -25697.521,E2 -25697.521} C_VEL
LIN {X 0,Y 143.359,Z 407.679,A -85,B 0,C 180,E1 -25699.711,E2 -25699.711} C_VEL
LIN {X 0,Y 141.125,Z 400.113,A -85,B 0,C 180,E1 -25703.302,E2 -25703.302} C_VEL
LIN {X 0,Y 138.179,Z 392.34,A -85,B 0,C 180,E1 -25707.395,E2 -25707.395} C_VEL
LIN {X 0,Y 136.417,Z 388.101,A -85,B 0,C 180,E1 -25709.847,E2 -25709.847} C_VEL
LIN {X 0,Y 134.208,Z 383.393,A -85,B 0,C 180,E1 -25712.897,E2 -25712.897} C_VEL
LIN {X 0,Y 131.88,Z 379.667,A -85,B 0,C 180,E1 -25716.025,E2 -25716.025} C_VEL
LIN {X 0,Y 131.029,Z 377.537,A -85,B 0,C 180,E1 -25717.532,E2 -25717.532} C_VEL
LIN {X 0,Y 128.152,Z 373.574,A -85,B 0,C 180,E1 -25722.136,E2 -25722.136} C_VEL
LIN {X 0,Y 127.223,Z 371.097,A -85,B 0,C 180,E1 -25724.377,E2 -25724.377} C_VEL
LIN {X 0,Y 124.006,Z 367.855,A -85,B 0,C 180,E1 -25732.834,E2 -25732.834} C_VEL
LIN {X 0,Y 123.391,Z 367.804,A -85,B 0,C 180,E1 -25735.553,E2 -25735.553} C_VEL
LIN {X 0,Y 122.813,Z 368.992,A -85,B 0,C 180,E1 -25738.259,E2 -25738.259} C_VEL
LIN {X 0,Y 122.058,Z 373.931,A -85,B 0,C 180,E1 -25745.476,E2 -25745.476} C_VEL
LIN {X 0,Y 122.289,Z 374.669,A -85,B 0,C 180,E1 -25747.342,E2 -25747.342} C_VEL
LIN {X 0,Y 124.931,Z 377.088,A -85,B 0,C 180,E1 -25755.394,E2 -25755.394} C_VEL
LIN {X 0,Y 125.781,Z 379.53,A -85,B 0,C 180,E1 -25757.899,E2 -25757.899} C_VEL
LIN {X 0,Y 128.289,Z 382.836,A -85,B 0,C 180,E1 -25762.55,E2 -25762.55} C_VEL
LIN {X 0,Y 131.343,Z 388.143,A -85,B 0,C 180,E1 -25767.615,E2 -25767.615} C_VEL
LIN {X 0,Y 133.082,Z 391.013,A -85,B 0,C 180,E1 -25770.112,E2 -25770.112} C_VEL
LIN {X 0,Y 135.839,Z 398.005,A -85,B 0,C 180,E1 -25774.689,E2 -25774.689} C_VEL
LIN {X 0,Y 137.917,Z 404.771,A -85,B 0,C 180,E1 -25778.553,E2 -25778.553} C_VEL
LIN {X 0,Y 139.052,Z 410.999,A -85,B 0,C 180,E1 -25781.737,E2 -25781.737} C_VEL
LIN {X 0,Y 139.24,Z 416.89,A -85,B 0,C 180,E1 -25784.437,E2 -25784.437} C_VEL
LIN {X 0,Y 138.489,Z 424.592,A -85,B 0,C 180,E1 -25787.891,E2 -25787.891} C_VEL
LIN {X 0,Y 138.254,Z 426.229,A -85,B 0,C 180,E1 -25788.639,E2 -25788.639} C_VEL
LIN {X 0,Y 136.724,Z 429.785,A -85,B 0,C 180,E1 -25790.021,E2 -25790.021} C_VEL
LIN {X 0,Y 132.194,Z 437.628,A -85,B 0,C 180,E1 -25793.267,E2 -25793.267} C_VEL
LIN {X 0,Y 127.213,Z 445.294,A -85,B 0,C 180,E1 -25797.411,E2 -25797.411} C_VEL
LIN {X 0,Y 122.06,Z 452.339,A -85,B 0,C 180,E1 -25802.575,E2 -25802.575} C_VEL
LIN {X 0,Y 118.601,Z 457.021,A -85,B 0,C 180,E1 -25807.348,E2 -25807.348} C_VEL
LIN {X 0,Y 115.848,Z 460.601,A -85,B 0,C 180,E1 -25812.344,E2 -25812.344} C_VEL
LIN {X 0,Y 114.499,Z 462.447,A -85,B 0,C 180,E1 -25815.789,E2 -25815.789} C_VEL
LIN {X 0,Y 113.514,Z 463.83,A -85,B 0,C 180,E1 -25819.298,E2 -25819.298} C_VEL
LIN {X 0,Y 112.424,Z 465.418,A -85,B 0,C 180,E1 -25826.418,E2 -25826.418} C_VEL
LIN {X 0,Y 112.335,Z 465.642,A -85,B 0,C 180,E1 -25830.002,E2 -25830.002} C_VEL
LIN {X 0,Y 112.425,Z 465.445,A -85,B 0,C 180,E1 -25833.586,E2 -25833.586} C_VEL
LIN {X 0,Y 113.509,Z 463.891,A -85,B 0,C 180,E1 -25840.706,E2 -25840.706} C_VEL
LIN {X 0,Y 114.499,Z 462.534,A -85,B 0,C 180,E1 -25844.214,E2 -25844.214} C_VEL
LIN {X 0,Y 116.627,Z 459.666,A -85,B 0,C 180,E1 -25849.357,E2 -25849.357} C_VEL
LIN {X 0,Y 119.634,Z 455.771,A -85,B 0,C 180,E1 -25854.283,E2 -25854.283} C_VEL
LIN {X 0,Y 123.38,Z 450.746,A -85,B 0,C 180,E1 -25858.96,E2 -25858.96} C_VEL
LIN {X 0,Y 127.946,Z 444.409,A -85,B 0,C 180,E1 -25863.319,E2 -25863.319} C_VEL
LIN {X 0,Y 132.747,Z 436.929,A -85,B 0,C 180,E1 -25867.222,E2 -25867.222} C_VEL
LIN {X 0,Y 137.579,Z 428.413,A -85,B 0,C 180,E1 -25870.642,E2 -25870.642} C_VEL
LIN {X 0,Y 138.287,Z 426.646,A -85,B 0,C 180,E1 -25871.353,E2 -25871.353} C_VEL
LIN {X 0,Y 139.135,Z 419.771,A -85,B 0,C 180,E1 -25874.481,E2 -25874.481} C_VEL
LIN {X 0,Y 139.324,Z 412.673,A -85,B 0,C 180,E1 -25877.661,E2 -25877.661} C_VEL
LIN {X 0,Y 138.41,Z 406.8,A -85,B 0,C 180,E1 -25880.599,E2 -25880.599} C_VEL
LIN {X 0,Y 136.468,Z 399.626,A -85,B 0,C 180,E1 -25884.594,E2 -25884.594} C_VEL
LIN {X 0,Y 133.702,Z 392.508,A -85,B 0,C 180,E1 -25889.169,E2 -25889.169} C_VEL
LIN {X 0,Y 130.866,Z 386.839,A -85,B 0,C 180,E1 -25893.667,E2 -25893.667} C_VEL
LIN {X 0,Y 129.327,Z 384.896,A -85,B 0,C 180,E1 -25895.947,E2 -25895.947} C_VEL
LIN {X 0,Y 127.689,Z 381.751,A -85,B 0,C 180,E1 -25899.039,E2 -25899.039} C_VEL
LIN {X 0,Y 125.525,Z 378.896,A -85,B 0,C 180,E1 -25903.325,E2 -25903.325} C_VEL
LIN {X 0,Y 124.932,Z 376.885,A -85,B 0,C 180,E1 -25905.336,E2 -25905.336} C_VEL
LIN {X 0,Y 122.084,Z 373.158,A -85,B 0,C 180,E1 -25920,E2 -25920} C_VEL
LIN {X 0,Y 123.904,Z 376.504,A -85,B 0,C 180,E1 -25931.451,E2 -25931.451} C_VEL
LIN {X 0,Y 125.264,Z 378.143,A -85,B 0,C 180,E1 -25934.936,E2 -25934.936} C_VEL
LIN {X 0,Y 126.784,Z 381.892,A -85,B 0,C 180,E1 -25938.796,E2 -25938.796} C_VEL
LIN {X 0,Y 128.195,Z 383.727,A -85,B 0,C 180,E1 -25941.253,E2 -25941.253} C_VEL
LIN {X 0,Y 129.556,Z 387.247,A -85,B 0,C 180,E1 -25944.007,E2 -25944.007} C_VEL
LIN {X 0,Y 130.991,Z 389.692,A -85,B 0,C 180,E1 -25946.237,E2 -25946.237} C_VEL
LIN {X 0,Y 133.242,Z 395.354,A -85,B 0,C 180,E1 -25950.072,E2 -25950.072} C_VEL
LIN {X 0,Y 135.5,Z 401.757,A -85,B 0,C 180,E1 -25953.914,E2 -25953.914} C_VEL
LIN {X 0,Y 137.539,Z 409.119,A -85,B 0,C 180,E1 -25957.82,E2 -25957.82} C_VEL
LIN {X 0,Y 138.498,Z 414.543,A -85,B 0,C 180,E1 -25960.432,E2 -25960.432} C_VEL
LIN {X 0,Y 138.264,Z 420.076,A -85,B 0,C 180,E1 -25962.652,E2 -25962.652} C_VEL
LIN {X 0,Y 136.911,Z 428.439,A -85,B 0,C 180,E1 -25965.944,E2 -25965.944} C_VEL
LIN {X 0,Y 134.889,Z 436.38,A -85,B 0,C 180,E1 -25969.362,E2 -25969.362} C_VEL
LIN {X 0,Y 133.512,Z 439.704,A -85,B 0,C 180,E1 -25970.826,E2 -25970.826} C_VEL
LIN {X 0,Y 128.238,Z 448.313,A -85,B 0,C 180,E1 -25974.868,E2 -25974.868} C_VEL
LIN {X 0,Y 123.666,Z 455.205,A -85,B 0,C 180,E1 -25979.237,E2 -25979.237} C_VEL
LIN {X 0,Y 119.653,Z 460.726,A -85,B 0,C 180,E1 -25983.862,E2 -25983.862} C_VEL
LIN {X 0,Y 116.429,Z 465.059,A -85,B 0,C 180,E1 -25988.765,E2 -25988.765} C_VEL
LIN {X 0,Y 114.871,Z 467.36,A -85,B 0,C 180,E1 -25992.186,E2 -25992.186} C_VEL
LIN {X 0,Y 113.666,Z 469.224,A -85,B 0,C 180,E1 -25995.68,E2 -25995.68} C_VEL
LIN {X 0,Y 112.34,Z 471.627,A -85,B 0,C 180,E1 -26002.811,E2 -26002.811} C_VEL
LIN {X 0,Y 112.137,Z 472.24,A -85,B 0,C 180,E1 -26006.405,E2 -26006.405} C_VEL
LIN {X 0,Y 112.261,Z 472.458,A -85,B 0,C 180,E1 -26009.998,E2 -26009.998} C_VEL
LIN {X 0,Y 112.137,Z 472.226,A -85,B 0,C 180,E1 -26013.592,E2 -26013.592} C_VEL
LIN {X 0,Y 112.34,Z 471.605,A -85,B 0,C 180,E1 -26017.186,E2 -26017.186} C_VEL
LIN {X 0,Y 113.664,Z 469.179,A -85,B 0,C 180,E1 -26024.317,E2 -26024.317} C_VEL
LIN {X 0,Y 115.596,Z 466.22,A -85,B 0,C 180,E1 -26029.533,E2 -26029.533} C_VEL
LIN {X 0,Y 118.487,Z 462.227,A -85,B 0,C 180,E1 -26034.53,E2 -26034.53} C_VEL
LIN {X 0,Y 122.936,Z 456.095,A -85,B 0,C 180,E1 -26040.012,E2 -26040.012} C_VEL
LIN {X 0,Y 127.369,Z 449.397,A -85,B 0,C 180,E1 -26044.44,E2 -26044.44} C_VEL
LIN {X 0,Y 132.539,Z 441.096,A -85,B 0,C 180,E1 -26048.537,E2 -26048.537} C_VEL
LIN {X 0,Y 134.265,Z 437.862,A -85,B 0,C 180,E1 -26049.88,E2 -26049.88} C_VEL
LIN {X 0,Y 136.461,Z 430.015,A -85,B 0,C 180,E1 -26053.299,E2 -26053.299} C_VEL
LIN {X 0,Y 137.987,Z 421.221,A -85,B 0,C 180,E1 -26056.818,E2 -26056.818} C_VEL
LIN {X 0,Y 138.486,Z 414.977,A -85,B 0,C 180,E1 -26059.249,E2 -26059.249} C_VEL
LIN {X 0,Y 137.81,Z 410.548,A -85,B 0,C 180,E1 -26061.324,E2 -26061.324} C_VEL
LIN {X 0,Y 135.808,Z 402.905,A -85,B 0,C 180,E1 -26065.302,E2 -26065.302} C_VEL
LIN {X 0,Y 133.545,Z 396.372,A -85,B 0,C 180,E1 -26069.129,E2 -26069.129} C_VEL
LIN {X 0,Y 132.704,Z 393.843,A -85,B 0,C 180,E1 -26070.667,E2 -26070.667} C_VEL
LIN {X 0,Y 130.364,Z 388.645,A -85,B 0,C 180,E1 -26074.451,E2 -26074.451} C_VEL
LIN {X 0,Y 127.771,Z 383.33,A -85,B 0,C 180,E1 -26079.053,E2 -26079.053} C_VEL
LIN {X 0,Y 125.514,Z 379.333,A -85,B 0,C 180,E1 -26083.637,E2 -26083.637} C_VEL
LIN {X 0,Y 124.953,Z 377.638,A -85,B 0,C 180,E1 -26085.339,E2 -26085.339} C_VEL
LIN {X 0,Y 122.41,Z 374.783,A -85,B 0,C 180,E1 -26092.992,E2 -26092.992} C_VEL
LIN {X 0,Y 121.892,Z 372.65,A -85,B 0,C 180,E1 -26100,E2 -26100} C_VEL
LIN {X 0,Y 122.289,Z 374.669,A -85,B 0,C 180,E1 -26107.342,E2 -26107.342} C_VEL
LIN {X 0,Y 122.518,Z 375.738,A -85,B 0,C 180,E1 -26109.111,E2 -26109.111} C_VEL
LIN {X 0,Y 122.514,Z 379.135,A -85,B 0,C 180,E1 -26111.78,E2 -26111.78} C_VEL
LIN {X 0,Y 122.492,Z 383.77,A -85,B 0,C 180,E1 -26114.935,E2 -26114.935} C_VEL
LIN {X 0,Y 122.713,Z 384.963,A -85,B 0,C 180,E1 -26116.069,E2 -26116.069} C_VEL
LIN {X 0,Y 125.001,Z 388.689,A -85,B 0,C 180,E1 -26121.436,E2 -26121.436} C_VEL
LIN {X 0,Y 127.361,Z 393.25,A -85,B 0,C 180,E1 -26126.197,E2 -26126.197} C_VEL
LIN {X 0,Y 129.194,Z 396.928,A -85,B 0,C 180,E1 -26129.502,E2 -26129.502} C_VEL
LIN {X 0,Y 131.704,Z 404.544,A -85,B 0,C 180,E1 -26134.767,E2 -26134.767} C_VEL
LIN {X 0,Y 133.063,Z 410.41,A -85,B 0,C 180,E1 -26138.335,E2 -26138.335} C_VEL
LIN {X 0,Y 133.628,Z 416.206,A -85,B 0,C 180,E1 -26141.462,E2 -26141.462} C_VEL
LIN {X 0,Y 133.211,Z 422.285,A -85,B 0,C 180,E1 -26144.397,E2 -26144.397} C_VEL
LIN {X 0,Y 132.169,Z 428.238,A -85,B 0,C 180,E1 -26147.317,E2 -26147.317} C_VEL
LIN {X 0,Y 129.374,Z 433.306,A -85,B 0,C 180,E1 -26149.32,E2 -26149.32} C_VEL
LIN {X 0,Y 123.922,Z 441.896,A -85,B 0,C 180,E1 -26153.455,E2 -26153.455} C_VEL
LIN {X 0,Y 118.831,Z 448.755,A -85,B 0,C 180,E1 -26157.842,E2 -26157.842} C_VEL
LIN {X 0,Y 114.488,Z 454.242,A -85,B 0,C 180,E1 -26162.589,E2 -26162.589} C_VEL
LIN {X 0,Y 110.99,Z 458.543,A -85,B 0,C 180,E1 -26167.673,E2 -26167.673} C_VEL
LIN {X 0,Y 109.11,Z 460.817,A -85,B 0,C 180,E1 -26171.215,E2 -26171.215} C_VEL
LIN {X 0,Y 107.623,Z 462.663,A -85,B 0,C 180,E1 -26174.86,E2 -26174.86} C_VEL
LIN {X 0,Y 106.533,Z 464.046,A -85,B 0,C 180,E1 -26178.587,E2 -26178.587} C_VEL
LIN {X 0,Y 105.777,Z 465.03,A -85,B 0,C 180,E1 -26182.366,E2 -26182.366} C_VEL
LIN {X 0,Y 105.266,Z 465.856,A -85,B 0,C 180,E1 -26190.002,E2 -26190.002} C_VEL
LIN {X 0,Y 105.344,Z 465.66,A -85,B 0,C 180,E1 -26193.827,E2 -26193.827} C_VEL
LIN {X 0,Y 105.776,Z 465.073,A -85,B 0,C 180,E1 -26197.638,E2 -26197.638} C_VEL
LIN {X 0,Y 106.528,Z 464.106,A -85,B 0,C 180,E1 -26201.417,E2 -26201.417} C_VEL
LIN {X 0,Y 107.622,Z 462.749,A -85,B 0,C 180,E1 -26205.143,E2 -26205.143} C_VEL
LIN {X 0,Y 109.945,Z 459.881,A -85,B 0,C 180,E1 -26210.585,E2 -26210.585} C_VEL
LIN {X 0,Y 113.178,Z 455.986,A -85,B 0,C 180,E1 -26215.766,E2 -26215.766} C_VEL
LIN {X 0,Y 117.223,Z 450.96,A -85,B 0,C 180,E1 -26220.639,E2 -26220.639} C_VEL
LIN {X 0,Y 122.073,Z 444.622,A -85,B 0,C 180,E1 -26225.151,E2 -26225.151} C_VEL
LIN {X 0,Y 126.852,Z 437.635,A -85,B 0,C 180,E1 -26228.932,E2 -26228.932} C_VEL
LIN {X 0,Y 132.172,Z 428.629,A -85,B 0,C 180,E1 -26232.685,E2 -26232.685} C_VEL
LIN {X 0,Y 133.25,Z 422.646,A -85,B 0,C 180,E1 -26235.637,E2 -26235.637} C_VEL
LIN {X 0,Y 133.724,Z 415.705,A -85,B 0,C 180,E1 -26238.996,E2 -26238.996} C_VEL
LIN {X 0,Y 133.165,Z 410.828,A -85,B 0,C 180,E1 -26241.674,E2 -26241.674} C_VEL
LIN {X 0,Y 131.566,Z 403.839,A -85,B 0,C 180,E1 -26245.93,E2 -26245.93} C_VEL
LIN {X 0,Y 129.289,Z 397.034,A -85,B 0,C 180,E1 -26250.71,E2 -26250.71} C_VEL
LIN {X 0,Y 126.746,Z 391.938,A -85,B 0,C 180,E1 -26255.425,E2 -26255.425} C_VEL
LIN {X 0,Y 124.457,Z 387.793,A -85,B 0,C 180,E1 -26260.195,E2 -26260.195} C_VEL
LIN {X 0,Y 123.079,Z 385.787,A -85,B 0,C 180,E1 -26263.411,E2 -26263.411} C_VEL
LIN {X 0,Y 122.155,Z 383.336,A -85,B 0,C 180,E1 -26266.695,E2 -26266.695} C_VEL
LIN {X 0,Y 120.209,Z 380.065,A -85,B 0,C 180,E1 -26280,E2 -26280} C_VEL
LIN {X 0,Y 121.574,Z 383.029,A -85,B 0,C 180,E1 -26290.659,E2 -26290.659} C_VEL
LIN {X 0,Y 122.44,Z 384.104,A -85,B 0,C 180,E1 -26293.273,E2 -26293.273} C_VEL
LIN {X 0,Y 124.006,Z 388.276,A -85,B 0,C 180,E1 -26298.162,E2 -26298.162} C_VEL
LIN {X 0,Y 125.211,Z 390.299,A -85,B 0,C 180,E1 -26300.729,E2 -26300.729} C_VEL
LIN {X 0,Y 127.324,Z 395.495,A -85,B 0,C 180,E1 -26305.327,E2 -26305.327} C_VEL
LIN {X 0,Y 129.274,Z 401.407,A -85,B 0,C 180,E1 -26309.559,E2 -26309.559} C_VEL
LIN {X 0,Y 131.003,Z 407.175,A -85,B 0,C 180,E1 -26313.276,E2 -26313.276} C_VEL
LIN {X 0,Y 132.542,Z 414.261,A -85,B 0,C 180,E1 -26317.309,E2 -26317.309} C_VEL
LIN {X 0,Y 132.975,Z 419.297,A -85,B 0,C 180,E1 -26319.854,E2 -26319.854} C_VEL
LIN {X 0,Y 131.541,Z 427.869,A -85,B 0,C 180,E1 -26323.456,E2 -26323.456} C_VEL
LIN {X 0,Y 129.267,Z 436.155,A -85,B 0,C 180,E1 -26327.187,E2 -26327.187} C_VEL
LIN {X 0,Y 128.01,Z 439.488,A -85,B 0,C 180,E1 -26328.789,E2 -26328.789} C_VEL
LIN {X 0,Y 122.47,Z 448.098,A -85,B 0,C 180,E1 -26332.946,E2 -26332.946} C_VEL
LIN {X 0,Y 117.572,Z 454.989,A -85,B 0,C 180,E1 -26337.453,E2 -26337.453} C_VEL
LIN {X 0,Y 113.284,Z 460.51,A -85,B 0,C 180,E1 -26342.27,E2 -26342.27} C_VEL
LIN {X 0,Y 109.821,Z 464.844,A -85,B 0,C 180,E1 -26347.419,E2 -26347.419} C_VEL
LIN {X 0,Y 108.087,Z 467.144,A -85,B 0,C 180,E1 -26351.026,E2 -26351.026} C_VEL
LIN {X 0,Y 106.772,Z 469.008,A -85,B 0,C 180,E1 -26354.733,E2 -26354.733} C_VEL
LIN {X 0,Y 105.283,Z 471.411,A -85,B 0,C 180,E1 -26362.326,E2 -26362.326} C_VEL
LIN {X 0,Y 105.046,Z 472.025,A -85,B 0,C 180,E1 -26366.162,E2 -26366.162} C_VEL
LIN {X 0,Y 105.173,Z 472.243,A -85,B 0,C 180,E1 -26369.998,E2 -26369.998} C_VEL
LIN {X 0,Y 105.046,Z 472.01,A -85,B 0,C 180,E1 -26373.834,E2 -26373.834} C_VEL
LIN {X 0,Y 105.282,Z 471.389,A -85,B 0,C 180,E1 -26377.67,E2 -26377.67} C_VEL
LIN {X 0,Y 106.771,Z 468.962,A -85,B 0,C 180,E1 -26385.264,E2 -26385.264} C_VEL
LIN {X 0,Y 108.896,Z 466.002,A -85,B 0,C 180,E1 -26390.789,E2 -26390.789} C_VEL
LIN {X 0,Y 112.05,Z 462.009,A -85,B 0,C 180,E1 -26396.041,E2 -26396.041} C_VEL
LIN {X 0,Y 116.829,Z 455.877,A -85,B 0,C 180,E1 -26401.758,E2 -26401.758} C_VEL
LIN {X 0,Y 121.541,Z 449.178,A -85,B 0,C 180,E1 -26406.346,E2 -26406.346} C_VEL
LIN {X 0,Y 127.047,Z 440.878,A -85,B 0,C 180,E1 -26410.538,E2 -26410.538} C_VEL
LIN {X 0,Y 128.634,Z 437.633,A -85,B 0,C 180,E1 -26412.009,E2 -26412.009} C_VEL
LIN {X 0,Y 131.079,Z 429.321,A -85,B 0,C 180,E1 -26415.812,E2 -26415.812} C_VEL
LIN {X 0,Y 132.545,Z 421.55,A -85,B 0,C 180,E1 -26419.106,E2 -26419.106} C_VEL
LIN {X 0,Y 132.867,Z 416.801,A -85,B 0,C 180,E1 -26421.18,E2 -26421.18} C_VEL
LIN {X 0,Y 131.545,Z 409.621,A -85,B 0,C 180,E1 -26425.147,E2 -26425.147} C_VEL
LIN {X 0,Y 129.83,Z 403.194,A -85,B 0,C 180,E1 -26429.054,E2 -26429.054} C_VEL
LIN {X 0,Y 128.301,Z 398.533,A -85,B 0,C 180,E1 -26432.25,E2 -26432.25} C_VEL
LIN {X 0,Y 126.768,Z 394.371,A -85,B 0,C 180,E1 -26435.43,E2 -26435.43} C_VEL
LIN {X 0,Y 124.572,Z 389.228,A -85,B 0,C 180,E1 -26440.214,E2 -26440.214} C_VEL
LIN {X 0,Y 123.195,Z 386.698,A -85,B 0,C 180,E1 -26443.427,E2 -26443.427} C_VEL
LIN {X 0,Y 122.728,Z 385.089,A -85,B 0,C 180,E1 -26445.067,E2 -26445.067} C_VEL
LIN {X 0,Y 122.223,Z 383.903,A -85,B 0,C 180,E1 -26446.703,E2 -26446.703} C_VEL
LIN {X 0,Y 120.408,Z 381.554,A -85,B 0,C 180,E1 -26453.296,E2 -26453.296} C_VEL
LIN {X 0,Y 120.029,Z 379.599,A -85,B 0,C 180,E1 -26460,E2 -26460} C_VEL
LIN {X 0,Y 121.869,Z 383.204,A -85,B 0,C 180,E1 -26473.337,E2 -26473.337} C_VEL
LIN {X 0,Y 122.432,Z 383.998,A -85,B 0,C 180,E1 -26474.97,E2 -26474.97} C_VEL
LIN {X 0,Y 122.713,Z 384.963,A -85,B 0,C 180,E1 -26476.069,E2 -26476.069} C_VEL
LIN {X 0,Y 123.234,Z 387.673,A -85,B 0,C 180,E1 -26478.518,E2 -26478.518} C_VEL
LIN {X 0,Y 123.57,Z 393.408,A -85,B 0,C 180,E1 -26482.287,E2 -26482.287} C_VEL
LIN {X 0,Y 123.865,Z 398.139,A -85,B 0,C 180,E1 -26485.275,E2 -26485.275} C_VEL
LIN {X 0,Y 124.895,Z 402.078,A -85,B 0,C 180,E1 -26488.426,E2 -26488.426} C_VEL
LIN {X 0,Y 126.838,Z 409.211,A -85,B 0,C 180,E1 -26493.788,E2 -26493.788} C_VEL
LIN {X 0,Y 127.845,Z 415.244,A -85,B 0,C 180,E1 -26497.741,E2 -26497.741} C_VEL
LIN {X 0,Y 128.012,Z 419.645,A -85,B 0,C 180,E1 -26500.311,E2 -26500.311} C_VEL
LIN {X 0,Y 127.188,Z 425.671,A -85,B 0,C 180,E1 -26503.464,E2 -26503.464} C_VEL
LIN {X 0,Y 126.093,Z 430.225,A -85,B 0,C 180,E1 -26505.84,E2 -26505.84} C_VEL
LIN {X 0,Y 121.425,Z 437.57,A -85,B 0,C 180,E1 -26509.006,E2 -26509.006} C_VEL
LIN {X 0,Y 116.401,Z 444.566,A -85,B 0,C 180,E1 -26512.862,E2 -26512.862} C_VEL
LIN {X 0,Y 111.24,Z 450.968,A -85,B 0,C 180,E1 -26517.522,E2 -26517.522} C_VEL
LIN {X 0,Y 106.89,Z 456.04,A -85,B 0,C 180,E1 -26522.599,E2 -26522.599} C_VEL
LIN {X 0,Y 103.369,Z 459.977,A -85,B 0,C 180,E1 -26528.043,E2 -26528.043} C_VEL
LIN {X 0,Y 100.791,Z 462.879,A -85,B 0,C 180,E1 -26533.807,E2 -26533.807} C_VEL
LIN {X 0,Y 99.575,Z 464.262,A -85,B 0,C 180,E1 -26537.778,E2 -26537.778} C_VEL
LIN {X 0,Y 98.754,Z 465.246,A -85,B 0,C 180,E1 -26541.819,E2 -26541.819} C_VEL
LIN {X 0,Y 98.192,Z 466.071,A -85,B 0,C 180,E1 -26550.002,E2 -26550.002} C_VEL
LIN {X 0,Y 98.754,Z 465.288,A -85,B 0,C 180,E1 -26558.185,E2 -26558.185} C_VEL
LIN {X 0,Y 100.789,Z 462.963,A -85,B 0,C 180,E1 -26566.197,E2 -26566.197} C_VEL
LIN {X 0,Y 103.328,Z 460.095,A -85,B 0,C 180,E1 -26571.97,E2 -26571.97} C_VEL
LIN {X 0,Y 106.808,Z 456.201,A -85,B 0,C 180,E1 -26577.427,E2 -26577.427} C_VEL
LIN {X 0,Y 111.18,Z 451.174,A -85,B 0,C 180,E1 -26582.502,E2 -26582.502} C_VEL
LIN {X 0,Y 116.338,Z 444.836,A -85,B 0,C 180,E1 -26587.165,E2 -26587.165} C_VEL
LIN {X 0,Y 122.195,Z 436.646,A -85,B 0,C 180,E1 -26591.609,E2 -26591.609} C_VEL
LIN {X 0,Y 126.042,Z 430.613,A -85,B 0,C 180,E1 -26594.187,E2 -26594.187} C_VEL
LIN {X 0,Y 127.059,Z 427.11,A -85,B 0,C 180,E1 -26595.978,E2 -26595.978} C_VEL
LIN {X 0,Y 128.023,Z 420.528,A -85,B 0,C 180,E1 -26599.438,E2 -26599.438} C_VEL
LIN {X 0,Y 127.967,Z 415.748,A -85,B 0,C 180,E1 -26602.184,E2 -26602.184} C_VEL
LIN {X 0,Y 126.926,Z 409.366,A -85,B 0,C 180,E1 -26606.378,E2 -26606.378} C_VEL
LIN {X 0,Y 125.567,Z 403.959,A -85,B 0,C 180,E1 -26610.332,E2 -26610.332} C_VEL
LIN {X 0,Y 123.607,Z 398.944,A -85,B 0,C 180,E1 -26614.938,E2 -26614.938} C_VEL
LIN {X 0,Y 121.671,Z 394.814,A -85,B 0,C 180,E1 -26619.722,E2 -26619.722} C_VEL
LIN {X 0,Y 119.625,Z 390.315,A -85,B 0,C 180,E1 -26626.408,E2 -26626.408} C_VEL
LIN {X 0,Y 118.031,Z 388.37,A -85,B 0,C 180,E1 -26633.16,E2 -26633.16} C_VEL
LIN {X 0,Y 117.934,Z 386.87,A -85,B 0,C 180,E1 -26640,E2 -26640} C_VEL
LIN {X 0,Y 119.005,Z 389.575,A -85,B 0,C 180,E1 -26650.205,E2 -26650.205} C_VEL
LIN {X 0,Y 119.894,Z 391.247,A -85,B 0,C 180,E1 -26653.56,E2 -26653.56} C_VEL
LIN {X 0,Y 121.915,Z 396.706,A -85,B 0,C 180,E1 -26660.236,E2 -26660.236} C_VEL
LIN {X 0,Y 123.409,Z 401.026,A -85,B 0,C 180,E1 -26664.33,E2 -26664.33} C_VEL
LIN {X 0,Y 124.901,Z 406.518,A -85,B 0,C 180,E1 -26668.573,E2 -26668.573} C_VEL
LIN {X 0,Y 126.084,Z 411.387,A -85,B 0,C 180,E1 -26671.976,E2 -26671.976} C_VEL
LIN {X 0,Y 127.249,Z 418.575,A -85,B 0,C 180,E1 -26676.422,E2 -26676.422} C_VEL
LIN {X 0,Y 127.321,Z 422.561,A -85,B 0,C 180,E1 -26678.594,E2 -26678.594} C_VEL
LIN {X 0,Y 125.5,Z 430.539,A -85,B 0,C 180,E1 -26682.222,E2 -26682.222} C_VEL
LIN {X 0,Y 123.201,Z 437.616,A -85,B 0,C 180,E1 -26685.668,E2 -26685.668} C_VEL
LIN {X 0,Y 121.741,Z 440.853,A -85,B 0,C 180,E1 -26687.287,E2 -26687.287} C_VEL
LIN {X 0,Y 115.927,Z 449.121,A -85,B 0,C 180,E1 -26691.581,E2 -26691.581} C_VEL
LIN {X 0,Y 110.838,Z 455.789,A -85,B 0,C 180,E1 -26696.3,E2 -26696.3} C_VEL
LIN {X 0,Y 105.703,Z 461.885,A -85,B 0,C 180,E1 -26702.261,E2 -26702.261} C_VEL
LIN {X 0,Y 102.266,Z 465.853,A -85,B 0,C 180,E1 -26707.79,E2 -26707.79} C_VEL
LIN {X 0,Y 99.898,Z 468.792,A -85,B 0,C 180,E1 -26713.654,E2 -26713.654} C_VEL
LIN {X 0,Y 98.871,Z 470.193,A -85,B 0,C 180,E1 -26717.686,E2 -26717.686} C_VEL
LIN {X 0,Y 98.251,Z 471.196,A -85,B 0,C 180,E1 -26721.773,E2 -26721.773} C_VEL
LIN {X 0,Y 97.952,Z 471.809,A -85,B 0,C 180,E1 -26725.884,E2 -26725.884} C_VEL
LIN {X 0,Y 98.077,Z 472.028,A -85,B 0,C 180,E1 -26729.998,E2 -26729.998} C_VEL
LIN {X 0,Y 98.25,Z 471.173,A -85,B 0,C 180,E1 -26738.223,E2 -26738.223} C_VEL
LIN {X 0,Y 98.87,Z 470.16,A -85,B 0,C 180,E1 -26742.311,E2 -26742.311} C_VEL
LIN {X 0,Y 99.897,Z 468.745,A -85,B 0,C 180,E1 -26746.342,E2 -26746.342} C_VEL
LIN {X 0,Y 102.264,Z 465.785,A -85,B 0,C 180,E1 -26752.206,E2 -26752.206} C_VEL
LIN {X 0,Y 105.7,Z 461.792,A -85,B 0,C 180,E1 -26757.736,E2 -26757.736} C_VEL
LIN {X 0,Y 110.819,Z 455.659,A -85,B 0,C 180,E1 -26763.702,E2 -26763.702} C_VEL
LIN {X 0,Y 115.85,Z 448.959,A -85,B 0,C 180,E1 -26768.446,E2 -26768.446} C_VEL
LIN {X 0,Y 121.697,Z 440.658,A -85,B 0,C 180,E1 -26772.728,E2 -26772.728} C_VEL
LIN {X 0,Y 123.783,Z 435.693,A -85,B 0,C 180,E1 -26775.208,E2 -26775.208} C_VEL
LIN {X 0,Y 126.038,Z 428.074,A -85,B 0,C 180,E1 -26778.831,E2 -26778.831} C_VEL
LIN {X 0,Y 127.357,Z 420.977,A -85,B 0,C 180,E1 -26782.051,E2 -26782.051} C_VEL
LIN {X 0,Y 126.738,Z 415.343,A -85,B 0,C 180,E1 -26785.362,E2 -26785.362} C_VEL
LIN {X 0,Y 125.416,Z 408.661,A -85,B 0,C 180,E1 -26789.713,E2 -26789.713} C_VEL
LIN {X 0,Y 123.825,Z 402.927,A -85,B 0,C 180,E1 -26793.995,E2 -26793.995} C_VEL
LIN {X 0,Y 122.951,Z 399.971,A -85,B 0,C 180,E1 -26796.414,E2 -26796.414} C_VEL
LIN {X 0,Y 121.145,Z 395.012,A -85,B 0,C 180,E1 -26801.393,E2 -26801.393} C_VEL
LIN {X 0,Y 119.72,Z 390.96,A -85,B 0,C 180,E1 -26806.419,E2 -26806.419} C_VEL
LIN {X 0,Y 118.773,Z 389.418,A -85,B 0,C 180,E1 -26809.775,E2 -26809.775} C_VEL
LIN {X 0,Y 117.787,Z 386.423,A -85,B 0,C 180,E1 -26820,E2 -26820} C_VEL
LIN {X 0,Y 119.4,Z 390.042,A -85,B 0,C 180,E1 -26833.618,E2 -26833.618} C_VEL
LIN {X 0,Y 120.787,Z 393.447,A -85,B 0,C 180,E1 -26838.664,E2 -26838.664} C_VEL
LIN {X 0,Y 121.487,Z 394.47,A -85,B 0,C 180,E1 -26840.31,E2 -26840.31} C_VEL
LIN {X 0,Y 123.475,Z 398.845,A -85,B 0,C 180,E1 -26845.27,E2 -26845.27} C_VEL
LIN {X 0,Y 124.895,Z 402.078,A -85,B 0,C 180,E1 -26848.426,E2 -26848.426} C_VEL
LIN {X 0,Y 125.511,Z 403.984,A -85,B 0,C 180,E1 -26849.977,E2 -26849.977} C_VEL
LIN {X 0,Y 125.694,Z 406.355,A -85,B 0,C 180,E1 -26851.413,E2 -26851.413} C_VEL
LIN {X 0,Y 125.33,Z 410.438,A -85,B 0,C 180,E1 -26853.392,E2 -26853.392} C_VEL
LIN {X 0,Y 123.626,Z 417.842,A -85,B 0,C 180,E1 -26856.565,E2 -26856.565} C_VEL
LIN {X 0,Y 122.305,Z 423.422,A -85,B 0,C 180,E1 -26859.322,E2 -26859.322} C_VEL
LIN {X 0,Y 120.749,Z 430.459,A -85,B 0,C 180,E1 -26863.322,E2 -26863.322} C_VEL
LIN {X 0,Y 120.038,Z 432.124,A -85,B 0,C 180,E1 -26864.178,E2 -26864.178} C_VEL
LIN {X 0,Y 113.763,Z 441.011,A -85,B 0,C 180,E1 -26868.389,E2 -26868.389} C_VEL
LIN {X 0,Y 107.985,Z 448.166,A -85,B 0,C 180,E1 -26872.988,E2 -26872.988} C_VEL
LIN {X 0,Y 103.621,Z 452.99,A -85,B 0,C 180,E1 -26877.143,E2 -26877.143} C_VEL
LIN {X 0,Y 99.288,Z 457.671,A -85,B 0,C 180,E1 -26882.609,E2 -26882.609} C_VEL
LIN {X 0,Y 95.761,Z 461.251,A -85,B 0,C 180,E1 -26888.474,E2 -26888.474} C_VEL
LIN {X 0,Y 93.982,Z 463.096,A -85,B 0,C 180,E1 -26892.597,E2 -26892.597} C_VEL
LIN {X 0,Y 92.654,Z 464.478,A -85,B 0,C 180,E1 -26896.849,E2 -26896.849} C_VEL
LIN {X 0,Y 91.731,Z 465.462,A -85,B 0,C 180,E1 -26901.188,E2 -26901.188} C_VEL
LIN {X 0,Y 91.114,Z 466.286,A -85,B 0,C 180,E1 -26910.002,E2 -26910.002} C_VEL
LIN {X 0,Y 91.207,Z 466.09,A -85,B 0,C 180,E1 -26914.421,E2 -26914.421} C_VEL
LIN {X 0,Y 91.731,Z 465.503,A -85,B 0,C 180,E1 -26918.816,E2 -26918.816} C_VEL
LIN {X 0,Y 92.651,Z 464.536,A -85,B 0,C 180,E1 -26923.155,E2 -26923.155} C_VEL
LIN {X 0,Y 93.978,Z 463.179,A -85,B 0,C 180,E1 -26927.407,E2 -26927.407} C_VEL
LIN {X 0,Y 96.785,Z 460.31,A -85,B 0,C 180,E1 -26933.541,E2 -26933.541} C_VEL
LIN {X 0,Y 100.542,Z 456.416,A -85,B 0,C 180,E1 -26939.296,E2 -26939.296} C_VEL
LIN {X 0,Y 105.27,Z 451.387,A -85,B 0,C 180,E1 -26944.576,E2 -26944.576} C_VEL
LIN {X 0,Y 110.763,Z 445.049,A -85,B 0,C 180,E1 -26949.385,E2 -26949.385} C_VEL
LIN {X 0,Y 116.564,Z 437.429,A -85,B 0,C 180,E1 -26953.654,E2 -26953.654} C_VEL
LIN {X 0,Y 119.963,Z 432.473,A -85,B 0,C 180,E1 -26955.863,E2 -26955.863} C_VEL
LIN {X 0,Y 120.802,Z 430.836,A -85,B 0,C 180,E1 -26956.655,E2 -26956.655} C_VEL
LIN {X 0,Y 122.39,Z 423.551,A -85,B 0,C 180,E1 -26960.828,E2 -26960.828} C_VEL
LIN {X 0,Y 122.493,Z 418.635,A -85,B 0,C 180,E1 -26963.978,E2 -26963.978} C_VEL
LIN {X 0,Y 121.652,Z 412.216,A -85,B 0,C 180,E1 -26968.671,E2 -26968.671} C_VEL
LIN {X 0,Y 120.735,Z 407.914,A -85,B 0,C 180,E1 -26972.245,E2 -26972.245} C_VEL
LIN {X 0,Y 119.577,Z 404.555,A -85,B 0,C 180,E1 -26975.706,E2 -26975.706} C_VEL
LIN {X 0,Y 117.927,Z 400.466,A -85,B 0,C 180,E1 -26980.866,E2 -26980.866} C_VEL
LIN {X 0,Y 116.59,Z 397.287,A -85,B 0,C 180,E1 -26986.047,E2 -26986.047} C_VEL
LIN {X 0,Y 115.89,Z 395.827,A -85,B 0,C 180,E1 -26989.518,E2 -26989.518} C_VEL
LIN {X 0,Y 115.255,Z 393.511,A -85,B 0,C 180,E1 -27000,E2 -27000} C_VEL
LIN {X 0,Y 116.221,Z 396.305,A -85,B 0,C 180,E1 -27010.452,E2 -27010.452} C_VEL
LIN {X 0,Y 116.599,Z 397.128,A -85,B 0,C 180,E1 -27012.179,E2 -27012.179} C_VEL
LIN {X 0,Y 118.159,Z 402.256,A -85,B 0,C 180,E1 -27019.095,E2 -27019.095} C_VEL
LIN {X 0,Y 119.309,Z 406.544,A -85,B 0,C 180,E1 -27023.429,E2 -27023.429} C_VEL
LIN {X 0,Y 120.423,Z 411.823,A -85,B 0,C 180,E1 -27027.832,E2 -27027.832} C_VEL
LIN {X 0,Y 121.229,Z 416.704,A -85,B 0,C 180,E1 -27031.45,E2 -27031.45} C_VEL
LIN {X 0,Y 121.862,Z 423.777,A -85,B 0,C 180,E1 -27036.156,E2 -27036.156} C_VEL
LIN {X 0,Y 121.363,Z 426.862,A -85,B 0,C 180,E1 -27037.782,E2 -27037.782} C_VEL
LIN {X 0,Y 119.012,Z 434.441,A -85,B 0,C 180,E1 -27041.545,E2 -27041.545} C_VEL
LIN {X 0,Y 116.5,Z 440.635,A -85,B 0,C 180,E1 -27044.859,E2 -27044.859} C_VEL
LIN {X 0,Y 110.423,Z 448.907,A -85,B 0,C 180,E1 -27049.278,E2 -27049.278} C_VEL
LIN {X 0,Y 104.952,Z 455.573,A -85,B 0,C 180,E1 -27054.13,E2 -27054.13} C_VEL
LIN {X 0,Y 99.438,Z 461.67,A -85,B 0,C 180,E1 -27060.346,E2 -27060.346} C_VEL
LIN {X 0,Y 95.714,Z 465.637,A -85,B 0,C 180,E1 -27066.179,E2 -27066.179} C_VEL
LIN {X 0,Y 93.07,Z 468.576,A -85,B 0,C 180,E1 -27072.417,E2 -27072.417} C_VEL
LIN {X 0,Y 91.219,Z 470.981,A -85,B 0,C 180,E1 -27081.134,E2 -27081.134} C_VEL
LIN {X 0,Y 90.882,Z 471.594,A -85,B 0,C 180,E1 -27085.563,E2 -27085.563} C_VEL
LIN {X 0,Y 90.975,Z 471.812,A -85,B 0,C 180,E1 -27089.998,E2 -27089.998} C_VEL
LIN {X 0,Y 90.881,Z 471.579,A -85,B 0,C 180,E1 -27094.433,E2 -27094.433} C_VEL
LIN {X 0,Y 91.218,Z 470.957,A -85,B 0,C 180,E1 -27098.862,E2 -27098.862} C_VEL
LIN {X 0,Y 91.914,Z 469.943,A -85,B 0,C 180,E1 -27103.259,E2 -27103.259} C_VEL
LIN {X 0,Y 93.068,Z 468.527,A -85,B 0,C 180,E1 -27107.579,E2 -27107.579} C_VEL
LIN {X 0,Y 95.712,Z 465.568,A -85,B 0,C 180,E1 -27113.817,E2 -27113.817} C_VEL
LIN {X 0,Y 99.435,Z 461.574,A -85,B 0,C 180,E1 -27119.651,E2 -27119.651} C_VEL
LIN {X 0,Y 104.958,Z 455.441,A -85,B 0,C 180,E1 -27125.864,E2 -27125.864} C_VEL
LIN {X 0,Y 110.342,Z 448.74,A -85,B 0,C 180,E1 -27130.754,E2 -27130.754} C_VEL
LIN {X 0,Y 115.491,Z 441.931,A -85,B 0,C 180,E1 -27134.409,E2 -27134.409} C_VEL
LIN {X 0,Y 117.183,Z 438.822,A -85,B 0,C 180,E1 -27136.026,E2 -27136.026} C_VEL
LIN {X 0,Y 119.912,Z 431.471,A -85,B 0,C 180,E1 -27139.856,E2 -27139.856} C_VEL
LIN {X 0,Y 121.811,Z 423.967,A -85,B 0,C 180,E1 -27143.562,E2 -27143.562} C_VEL
LIN {X 0,Y 121.362,Z 418.105,A -85,B 0,C 180,E1 -27147.411,E2 -27147.411} C_VEL
LIN {X 0,Y 120.322,Z 411.583,A -85,B 0,C 180,E1 -27152.142,E2 -27152.142} C_VEL
LIN {X 0,Y 118.923,Z 405.415,A -85,B 0,C 180,E1 -27157.41,E2 -27157.41} C_VEL
LIN {X 0,Y 117.992,Z 402.054,A -85,B 0,C 180,E1 -27160.877,E2 -27160.877} C_VEL
LIN {X 0,Y 116.721,Z 398.095,A -85,B 0,C 180,E1 -27166.063,E2 -27166.063} C_VEL
LIN {X 0,Y 116.01,Z 396.126,A -85,B 0,C 180,E1 -27169.529,E2 -27169.529} C_VEL
LIN {X 0,Y 115.135,Z 393.073,A -85,B 0,C 180,E1 -27180,E2 -27180} C_VEL
LIN {X 0,Y 115.671,Z 395.586,A -85,B 0,C 180,E1 -27190.503,E2 -27190.503} C_VEL
LIN {X 0,Y 116.424,Z 396.959,A -85,B 0,C 180,E1 -27193.973,E2 -27193.973} C_VEL
LIN {X 0,Y 117.752,Z 400.153,A -85,B 0,C 180,E1 -27199.164,E2 -27199.164} C_VEL
LIN {X 0,Y 119.384,Z 404.306,A -85,B 0,C 180,E1 -27204.336,E2 -27204.336} C_VEL
LIN {X 0,Y 120.589,Z 407.603,A -85,B 0,C 180,E1 -27207.791,E2 -27207.791} C_VEL
LIN {X 0,Y 121.823,Z 413.588,A -85,B 0,C 180,E1 -27212.656,E2 -27212.656} C_VEL
LIN {X 0,Y 122.437,Z 419.008,A -85,B 0,C 180,E1 -27216.528,E2 -27216.528} C_VEL
LIN {X 0,Y 122.305,Z 423.422,A -85,B 0,C 180,E1 -27219.322,E2 -27219.322} C_VEL
LIN {X 0,Y 121.452,Z 426.099,A -85,B 0,C 180,E1 -27220.638,E2 -27220.638} C_VEL
LIN {X 0,Y 119.945,Z 428.899,A -85,B 0,C 180,E1 -27221.759,E2 -27221.759} C_VEL
LIN {X 0,Y 116.842,Z 433.107,A -85,B 0,C 180,E1 -27223.202,E2 -27223.202} C_VEL
LIN {X 0,Y 108.007,Z 442.257,A -85,B 0,C 180,E1 -27226.62,E2 -27226.62} C_VEL
LIN {X 0,Y 105.773,Z 444.6,A -85,B 0,C 180,E1 -27227.945,E2 -27227.945} C_VEL
LIN {X 0,Y 99.566,Z 451.401,A -85,B 0,C 180,E1 -27233.134,E2 -27233.134} C_VEL
LIN {X 0,Y 94.474,Z 456.475,A -85,B 0,C 180,E1 -27238.621,E2 -27238.621} C_VEL
LIN {X 0,Y 90.368,Z 460.409,A -85,B 0,C 180,E1 -27244.679,E2 -27244.679} C_VEL
LIN {X 0,Y 87.231,Z 463.312,A -85,B 0,C 180,E1 -27251.202,E2 -27251.202} C_VEL
LIN {X 0,Y 85.75,Z 464.694,A -85,B 0,C 180,E1 -27255.769,E2 -27255.769} C_VEL
LIN {X 0,Y 84.739,Z 465.677,A -85,B 0,C 180,E1 -27260.454,E2 -27260.454} C_VEL
LIN {X 0,Y 84.024,Z 466.501,A -85,B 0,C 180,E1 -27270.002,E2 -27270.002} C_VEL
LIN {X 0,Y 84.739,Z 465.718,A -85,B 0,C 180,E1 -27279.55,E2 -27279.55} C_VEL
LIN {X 0,Y 87.226,Z 463.394,A -85,B 0,C 180,E1 -27288.803,E2 -27288.803} C_VEL
LIN {X 0,Y 90.311,Z 460.525,A -85,B 0,C 180,E1 -27295.343,E2 -27295.343} C_VEL
LIN {X 0,Y 94.4,Z 456.631,A -85,B 0,C 180,E1 -27301.411,E2 -27301.411} C_VEL
LIN {X 0,Y 99.516,Z 451.601,A -85,B 0,C 180,E1 -27306.892,E2 -27306.892} C_VEL
LIN {X 0,Y 105.368,Z 445.263,A -85,B 0,C 180,E1 -27311.837,E2 -27311.837} C_VEL
LIN {X 0,Y 111.94,Z 437.093,A -85,B 0,C 180,E1 -27316.44,E2 -27316.44} C_VEL
LIN {X 0,Y 115.011,Z 432.692,A -85,B 0,C 180,E1 -27318.467,E2 -27318.467} C_VEL
LIN {X 0,Y 116.75,Z 426.477,A -85,B 0,C 180,E1 -27322.325,E2 -27322.325} C_VEL
LIN {X 0,Y 117.06,Z 422.367,A -85,B 0,C 180,E1 -27325.224,E2 -27325.224} C_VEL
LIN {X 0,Y 116.742,Z 417.474,A -85,B 0,C 180,E1 -27329.14,E2 -27329.14} C_VEL
LIN {X 0,Y 116.157,Z 413.127,A -85,B 0,C 180,E1 -27333.013,E2 -27333.013} C_VEL
LIN {X 0,Y 115.449,Z 410.477,A -85,B 0,C 180,E1 -27335.943,E2 -27335.943} C_VEL
LIN {X 0,Y 113.968,Z 405.983,A -85,B 0,C 180,E1 -27342.041,E2 -27342.041} C_VEL
LIN {X 0,Y 113.208,Z 403.965,A -85,B 0,C 180,E1 -27345.622,E2 -27345.622} C_VEL
LIN {X 0,Y 112.671,Z 402.341,A -85,B 0,C 180,E1 -27349.214,E2 -27349.214} C_VEL
LIN {X 0,Y 112.22,Z 399.985,A -85,B 0,C 180,E1 -27360,E2 -27360} C_VEL
LIN {X 0,Y 112.455,Z 401.7,A -85,B 0,C 180,E1 -27367.18,E2 -27367.18} C_VEL
LIN {X 0,Y 113.062,Z 402.868,A -85,B 0,C 180,E1 -27370.747,E2 -27370.747} C_VEL
LIN {X 0,Y 114.182,Z 407.675,A -85,B 0,C 180,E1 -27377.924,E2 -27377.924} C_VEL
LIN {X 0,Y 115.005,Z 412.068,A -85,B 0,C 180,E1 -27382.666,E2 -27382.666} C_VEL
LIN {X 0,Y 115.707,Z 417.003,A -85,B 0,C 180,E1 -27387.1,E2 -27387.1} C_VEL
LIN {X 0,Y 116.141,Z 422.075,A -85,B 0,C 180,E1 -27391.104,E2 -27391.104} C_VEL
LIN {X 0,Y 116.253,Z 427.296,A -85,B 0,C 180,E1 -27394.883,E2 -27394.883} C_VEL
LIN {X 0,Y 114.927,Z 431.835,A -85,B 0,C 180,E1 -27397.346,E2 -27397.346} C_VEL
LIN {X 0,Y 112.087,Z 438.815,A -85,B 0,C 180,E1 -27401.199,E2 -27401.199} C_VEL
LIN {X 0,Y 110.499,Z 441.916,A -85,B 0,C 180,E1 -27402.993,E2 -27402.993} C_VEL
LIN {X 0,Y 104.081,Z 449.929,A -85,B 0,C 180,E1 -27407.526,E2 -27407.526} C_VEL
LIN {X 0,Y 98.373,Z 456.353,A -85,B 0,C 180,E1 -27412.607,E2 -27412.607} C_VEL
LIN {X 0,Y 93.29,Z 461.454,A -85,B 0,C 180,E1 -27418.172,E2 -27418.172} C_VEL
LIN {X 0,Y 89.227,Z 465.422,A -85,B 0,C 180,E1 -27424.327,E2 -27424.327} C_VEL
LIN {X 0,Y 86.3,Z 468.36,A -85,B 0,C 180,E1 -27430.987,E2 -27430.987} C_VEL
LIN {X 0,Y 84.192,Z 470.765,A -85,B 0,C 180,E1 -27440.387,E2 -27440.387} C_VEL
LIN {X 0,Y 83.799,Z 471.379,A -85,B 0,C 180,E1 -27445.187,E2 -27445.187} C_VEL
LIN {X 0,Y 83.881,Z 471.597,A -85,B 0,C 180,E1 -27449.998,E2 -27449.998} C_VEL
LIN {X 0,Y 83.799,Z 471.363,A -85,B 0,C 180,E1 -27454.809,E2 -27454.809} C_VEL
LIN {X 0,Y 84.191,Z 470.74,A -85,B 0,C 180,E1 -27459.608,E2 -27459.608} C_VEL
LIN {X 0,Y 84.998,Z 469.727,A -85,B 0,C 180,E1 -27464.36,E2 -27464.36} C_VEL
LIN {X 0,Y 86.298,Z 468.31,A -85,B 0,C 180,E1 -27469.009,E2 -27469.009} C_VEL
LIN {X 0,Y 89.224,Z 465.35,A -85,B 0,C 180,E1 -27475.669,E2 -27475.669} C_VEL
LIN {X 0,Y 93.287,Z 461.356,A -85,B 0,C 180,E1 -27481.825,E2 -27481.825} C_VEL
LIN {X 0,Y 99.259,Z 455.222,A -85,B 0,C 180,E1 -27488.28,E2 -27488.28} C_VEL
LIN {X 0,Y 105.03,Z 448.521,A -85,B 0,C 180,E1 -27493.301,E2 -27493.301} C_VEL
LIN {X 0,Y 110.435,Z 441.709,A -85,B 0,C 180,E1 -27497.038,E2 -27497.038} C_VEL
LIN {X 0,Y 113.251,Z 435.821,A -85,B 0,C 180,E1 -27500.396,E2 -27500.396} C_VEL
LIN {X 0,Y 115.867,Z 428.453,A -85,B 0,C 180,E1 -27504.317,E2 -27504.317} C_VEL
LIN {X 0,Y 116.225,Z 426.992,A -85,B 0,C 180,E1 -27505.134,E2 -27505.134} C_VEL
LIN {X 0,Y 115.995,Z 420.856,A -85,B 0,C 180,E1 -27509.617,E2 -27509.617} C_VEL
LIN {X 0,Y 115.481,Z 415.633,A -85,B 0,C 180,E1 -27513.818,E2 -27513.818} C_VEL
LIN {X 0,Y 114.684,Z 410.704,A -85,B 0,C 180,E1 -27518.427,E2 -27518.427} C_VEL
LIN {X 0,Y 114.025,Z 407.471,A -85,B 0,C 180,E1 -27522.051,E2 -27522.051} C_VEL
LIN {X 0,Y 113.081,Z 403.726,A -85,B 0,C 180,E1 -27527.436,E2 -27527.436} C_VEL
LIN {X 0,Y 112.82,Z 402.784,A -85,B 0,C 180,E1 -27529.229,E2 -27529.229} C_VEL
LIN {X 0,Y 112.283,Z 401.45,A -85,B 0,C 180,E1 -27532.809,E2 -27532.809} C_VEL
LIN {X 0,Y 112.114,Z 399.575,A -85,B 0,C 180,E1 -27540,E2 -27540} C_VEL
LIN {X 0,Y 112.487,Z 402.089,A -85,B 0,C 180,E1 -27550.803,E2 -27550.803} C_VEL
LIN {X 0,Y 113.282,Z 404.583,A -85,B 0,C 180,E1 -27555.924,E2 -27555.924} C_VEL
LIN {X 0,Y 114.186,Z 406.908,A -85,B 0,C 180,E1 -27559.787,E2 -27559.787} C_VEL
LIN {X 0,Y 115.532,Z 411.209,A -85,B 0,C 180,E1 -27565.203,E2 -27565.203} C_VEL
LIN {X 0,Y 116.169,Z 413.874,A -85,B 0,C 180,E1 -27567.961,E2 -27567.961} C_VEL
LIN {X 0,Y 116.863,Z 419.456,A -85,B 0,C 180,E1 -27572.769,E2 -27572.769} C_VEL
LIN {X 0,Y 116.959,Z 423.511,A -85,B 0,C 180,E1 -27575.865,E2 -27575.865} C_VEL
LIN {X 0,Y 116.467,Z 427.201,A -85,B 0,C 180,E1 -27578.333,E2 -27578.333} C_VEL
LIN {X 0,Y 114.972,Z 432.353,A -85,B 0,C 180,E1 -27581.515,E2 -27581.515} C_VEL
LIN {X 0,Y 113.118,Z 435.303,A -85,B 0,C 180,E1 -27582.903,E2 -27582.903} C_VEL
LIN {X 0,Y 106.492,Z 443.775,A -85,B 0,C 180,E1 -27587.436,E2 -27587.436} C_VEL
LIN {X 0,Y 105.773,Z 444.6,A -85,B 0,C 180,E1 -27587.945,E2 -27587.945} C_VEL
LIN {X 0,Y 102.369,Z 447.861,A -85,B 0,C 180,E1 -27589.912,E2 -27589.912} C_VEL
LIN {X 0,Y 95.514,Z 452.689,A -85,B 0,C 180,E1 -27592.989,E2 -27592.989} C_VEL
LIN {X 0,Y 88.84,Z 456.862,A -85,B 0,C 180,E1 -27596.744,E2 -27596.744} C_VEL
LIN {X 0,Y 85.86,Z 459.011,A -85,B 0,C 180,E1 -27599.765,E2 -27599.765} C_VEL
LIN {X 0,Y 82.722,Z 461.683,A -85,B 0,C 180,E1 -27604.865,E2 -27604.865} C_VEL
LIN {X 0,Y 80.55,Z 463.528,A -85,B 0,C 180,E1 -27609.577,E2 -27609.577} C_VEL
LIN {X 0,Y 77.746,Z 465.893,A -85,B 0,C 180,E1 -27619.587,E2 -27619.587} C_VEL
LIN {X 0,Y 76.925,Z 466.716,A -85,B 0,C 180,E1 -27630.002,E2 -27630.002} C_VEL
LIN {X 0,Y 77.072,Z 466.52,A -85,B 0,C 180,E1 -27635.234,E2 -27635.234} C_VEL
LIN {X 0,Y 77.747,Z 465.933,A -85,B 0,C 180,E1 -27640.418,E2 -27640.418} C_VEL
LIN {X 0,Y 80.544,Z 463.608,A -85,B 0,C 180,E1 -27650.43,E2 -27650.43} C_VEL
LIN {X 0,Y 83.949,Z 460.739,A -85,B 0,C 180,E1 -27657.418,E2 -27657.418} C_VEL
LIN {X 0,Y 88.406,Z 456.845,A -85,B 0,C 180,E1 -27663.814,E2 -27663.814} C_VEL
LIN {X 0,Y 93.934,Z 451.815,A -85,B 0,C 180,E1 -27669.493,E2 -27669.493} C_VEL
LIN {X 0,Y 100.185,Z 445.476,A -85,B 0,C 180,E1 -27674.549,E2 -27674.549} C_VEL
LIN {X 0,Y 106.963,Z 437.557,A -85,B 0,C 180,E1 -27679.077,E2 -27679.077} C_VEL
LIN {X 0,Y 109.284,Z 434.521,A -85,B 0,C 180,E1 -27680.509,E2 -27680.509} C_VEL
LIN {X 0,Y 111.056,Z 429.532,A -85,B 0,C 180,E1 -27683.828,E2 -27683.828} C_VEL
LIN {X 0,Y 111.585,Z 425.407,A -85,B 0,C 180,E1 -27687.072,E2 -27687.072} C_VEL
LIN {X 0,Y 111.521,Z 420.066,A -85,B 0,C 180,E1 -27691.919,E2 -27691.919} C_VEL
LIN {X 0,Y 111.385,Z 418.169,A -85,B 0,C 180,E1 -27693.789,E2 -27693.789} C_VEL
LIN {X 0,Y 110.378,Z 413.722,A -85,B 0,C 180,E1 -27699.5,E2 -27699.5} C_VEL
LIN {X 0,Y 109.498,Z 410.397,A -85,B 0,C 180,E1 -27705.123,E2 -27705.123} C_VEL
LIN {X 0,Y 109.066,Z 408.69,A -85,B 0,C 180,E1 -27708.854,E2 -27708.854} C_VEL
LIN {X 0,Y 108.577,Z 406.927,A -85,B 0,C 180,E1 -27716.289,E2 -27716.289} C_VEL
LIN {X 0,Y 108.836,Z 406.284,A -85,B 0,C 180,E1 -27720,E2 -27720} C_VEL
LIN {X 0,Y 108.988,Z 407.997,A -85,B 0,C 180,E1 -27727.41,E2 -27727.41} C_VEL
LIN {X 0,Y 109.435,Z 409.331,A -85,B 0,C 180,E1 -27731.108,E2 -27731.108} C_VEL
LIN {X 0,Y 109.939,Z 412.801,A -85,B 0,C 180,E1 -27736.482,E2 -27736.482} C_VEL
LIN {X 0,Y 110.37,Z 416.031,A -85,B 0,C 180,E1 -27740.501,E2 -27740.501} C_VEL
LIN {X 0,Y 110.788,Z 421.989,A -85,B 0,C 180,E1 -27746.363,E2 -27746.363} C_VEL
LIN {X 0,Y 110.768,Z 427.99,A -85,B 0,C 180,E1 -27751.426,E2 -27751.426} C_VEL
LIN {X 0,Y 110.648,Z 430.174,A -85,B 0,C 180,E1 -27753.162,E2 -27753.162} C_VEL
LIN {X 0,Y 109.37,Z 433.818,A -85,B 0,C 180,E1 -27755.333,E2 -27755.333} C_VEL
LIN {X 0,Y 105.579,Z 441.693,A -85,B 0,C 180,E1 -27760.046,E2 -27760.046} C_VEL
LIN {X 0,Y 102.279,Z 445.924,A -85,B 0,C 180,E1 -27762.38,E2 -27762.38} C_VEL
LIN {X 0,Y 95.617,Z 453.212,A -85,B 0,C 180,E1 -27767.308,E2 -27767.308} C_VEL
LIN {X 0,Y 90.872,Z 457.959,A -85,B 0,C 180,E1 -27771.776,E2 -27771.776} C_VEL
LIN {X 0,Y 85.722,Z 462.674,A -85,B 0,C 180,E1 -27777.796,E2 -27777.796} C_VEL
LIN {X 0,Y 81.604,Z 466.28,A -85,B 0,C 180,E1 -27784.492,E2 -27784.492} C_VEL
LIN {X 0,Y 79.6,Z 468.145,A -85,B 0,C 180,E1 -27789.317,E2 -27789.317} C_VEL
LIN {X 0,Y 77.196,Z 470.55,A -85,B 0,C 180,E1 -27799.507,E2 -27799.507} C_VEL
LIN {X 0,Y 76.738,Z 471.164,A -85,B 0,C 180,E1 -27804.743,E2 -27804.743} C_VEL
LIN {X 0,Y 76.779,Z 471.381,A -85,B 0,C 180,E1 -27809.998,E2 -27809.998} C_VEL
LIN {X 0,Y 76.737,Z 471.148,A -85,B 0,C 180,E1 -27815.252,E2 -27815.252} C_VEL
LIN {X 0,Y 77.195,Z 470.524,A -85,B 0,C 180,E1 -27820.489,E2 -27820.489} C_VEL
LIN {X 0,Y 78.128,Z 469.511,A -85,B 0,C 180,E1 -27825.653,E2 -27825.653} C_VEL
LIN {X 0,Y 79.598,Z 468.093,A -85,B 0,C 180,E1 -27830.679,E2 -27830.679} C_VEL
LIN {X 0,Y 82.855,Z 465.133,A -85,B 0,C 180,E1 -27837.806,E2 -27837.806} C_VEL
LIN {X 0,Y 87.295,Z 461.138,A -85,B 0,C 180,E1 -27844.299,E2 -27844.299} C_VEL
LIN {X 0,Y 93.744,Z 455.003,A -85,B 0,C 180,E1 -27850.991,E2 -27850.991} C_VEL
LIN {X 0,Y 99.971,Z 448.303,A -85,B 0,C 180,E1 -27856.099,E2 -27856.099} C_VEL
LIN {X 0,Y 104.549,Z 442.984,A -85,B 0,C 180,E1 -27859.13,E2 -27859.13} C_VEL
LIN {X 0,Y 106.367,Z 439.972,A -85,B 0,C 180,E1 -27860.924,E2 -27860.924} C_VEL
LIN {X 0,Y 109.742,Z 432.512,A -85,B 0,C 180,E1 -27865.308,E2 -27865.308} C_VEL
LIN {X 0,Y 110.613,Z 429.854,A -85,B 0,C 180,E1 -27866.89,E2 -27866.89} C_VEL
LIN {X 0,Y 110.736,Z 424.102,A -85,B 0,C 180,E1 -27871.578,E2 -27871.578} C_VEL
LIN {X 0,Y 110.479,Z 418.639,A -85,B 0,C 180,E1 -27876.587,E2 -27876.587} C_VEL
LIN {X 0,Y 110.227,Z 415.848,A -85,B 0,C 180,E1 -27879.471,E2 -27879.471} C_VEL
LIN {X 0,Y 109.536,Z 411.538,A -85,B 0,C 180,E1 -27885.129,E2 -27885.129} C_VEL
LIN {X 0,Y 109.222,Z 409.211,A -85,B 0,C 180,E1 -27888.87,E2 -27888.87} C_VEL
LIN {X 0,Y 108.826,Z 407.78,A -85,B 0,C 180,E1 -27892.579,E2 -27892.579} C_VEL
LIN {X 0,Y 108.741,Z 405.9,A -85,B 0,C 180,E1 -27900,E2 -27900} C_VEL
LIN {X 0,Y 108.548,Z 407.545,A -85,B 0,C 180,E1 -27907.953,E2 -27907.953} C_VEL
LIN {X 0,Y 108.898,Z 408.437,A -85,B 0,C 180,E1 -27911.164,E2 -27911.164} C_VEL
LIN {X 0,Y 109.402,Z 410.492,A -85,B 0,C 180,E1 -27915.517,E2 -27915.517} C_VEL
LIN {X 0,Y 110.223,Z 413.462,A -85,B 0,C 180,E1 -27920.53,E2 -27920.53} C_VEL
LIN {X 0,Y 111.236,Z 417.921,A -85,B 0,C 180,E1 -27926.249,E2 -27926.249} C_VEL
LIN {X 0,Y 111.553,Z 423.503,A -85,B 0,C 180,E1 -27931.554,E2 -27931.554} C_VEL
LIN {X 0,Y 111.344,Z 427.465,A -85,B 0,C 180,E1 -27934.864,E2 -27934.864} C_VEL
LIN {X 0,Y 110.469,Z 431.028,A -85,B 0,C 180,E1 -27937.396,E2 -27937.396} C_VEL
LIN {X 0,Y 109.298,Z 434.184,A -85,B 0,C 180,E1 -27939.505,E2 -27939.505} C_VEL
LIN {X 0,Y 103.567,Z 441.447,A -85,B 0,C 180,E1 -27943.16,E2 -27943.16} C_VEL
LIN {X 0,Y 97.039,Z 448.6,A -85,B 0,C 180,E1 -27947.942,E2 -27947.942} C_VEL
LIN {X 0,Y 92.034,Z 453.424,A -85,B 0,C 180,E1 -27952.348,E2 -27952.348} C_VEL
LIN {X 0,Y 86.908,Z 458.105,A -85,B 0,C 180,E1 -27958.292,E2 -27958.292} C_VEL
LIN {X 0,Y 85.86,Z 459.011,A -85,B 0,C 180,E1 -27959.765,E2 -27959.765} C_VEL
LIN {X 0,Y 83.087,Z 460.961,A -85,B 0,C 180,E1 -27963.045,E2 -27963.045} C_VEL
LIN {X 0,Y 77.392,Z 463.633,A -85,B 0,C 180,E1 -27968.517,E2 -27968.517} C_VEL
LIN {X 0,Y 73.148,Z 465.202,A -85,B 0,C 180,E1 -27973.509,E2 -27973.509} C_VEL
LIN {X 0,Y 71.009,Z 466.011,A -85,B 0,C 180,E1 -27977.862,E2 -27977.862} C_VEL
LIN {X 0,Y 70.624,Z 466.202,A -85,B 0,C 180,E1 -27979.423,E2 -27979.423} C_VEL
LIN {X 0,Y 69.854,Z 466.931,A -85,B 0,C 180,E1 -27990.003,E2 -27990.003} C_VEL
LIN {X 0,Y 70.79,Z 466.148,A -85,B 0,C 180,E1 -28001.455,E2 -28001.455} C_VEL
LIN {X 0,Y 73.916,Z 463.824,A -85,B 0,C 180,E1 -28012.356,E2 -28012.356} C_VEL
LIN {X 0,Y 77.702,Z 460.954,A -85,B 0,C 180,E1 -28019.834,E2 -28019.834} C_VEL
LIN {X 0,Y 82.59,Z 457.06,A -85,B 0,C 180,E1 -28026.562,E2 -28026.562} C_VEL
LIN {X 0,Y 88.562,Z 452.029,A -85,B 0,C 180,E1 -28032.419,E2 -28032.419} C_VEL
LIN {X 0,Y 95.249,Z 445.69,A -85,B 0,C 180,E1 -28037.55,E2 -28037.55} C_VEL
LIN {X 0,Y 102.452,Z 437.77,A -85,B 0,C 180,E1 -28042.079,E2 -28042.079} C_VEL
LIN {X 0,Y 103.676,Z 436.292,A -85,B 0,C 180,E1 -28042.798,E2 -28042.798} C_VEL
LIN {X 0,Y 105.452,Z 432.358,A -85,B 0,C 180,E1 -28045.585,E2 -28045.585} C_VEL
LIN {X 0,Y 106.024,Z 429.57,A -85,B 0,C 180,E1 -28047.974,E2 -28047.974} C_VEL
LIN {X 0,Y 106.367,Z 425.032,A -85,B 0,C 180,E1 -28052.45,E2 -28052.45} C_VEL
LIN {X 0,Y 106.414,Z 423.048,A -85,B 0,C 180,E1 -28054.577,E2 -28054.577} C_VEL
LIN {X 0,Y 106.09,Z 420.448,A -85,B 0,C 180,E1 -28058.04,E2 -28058.04} C_VEL
LIN {X 0,Y 105.391,Z 416.606,A -85,B 0,C 180,E1 -28064.529,E2 -28064.529} C_VEL
LIN {X 0,Y 105.094,Z 414.877,A -85,B 0,C 180,E1 -28068.426,E2 -28068.426} C_VEL
LIN {X 0,Y 104.843,Z 413.706,A -85,B 0,C 180,E1 -28072.295,E2 -28072.295} C_VEL
LIN {X 0,Y 105.09,Z 412.369,A -85,B 0,C 180,E1 -28080,E2 -28080} C_VEL
LIN {X 0,Y 105.126,Z 414.122,A -85,B 0,C 180,E1 -28087.684,E2 -28087.684} C_VEL
LIN {X 0,Y 105.358,Z 415.734,A -85,B 0,C 180,E1 -28091.544,E2 -28091.544} C_VEL
LIN {X 0,Y 105.554,Z 418.055,A -85,B 0,C 180,E1 -28095.446,E2 -28095.446} C_VEL
LIN {X 0,Y 105.715,Z 420.987,A -85,B 0,C 180,E1 -28099.415,E2 -28099.415} C_VEL
LIN {X 0,Y 105.659,Z 425.737,A -85,B 0,C 180,E1 -28104.565,E2 -28104.565} C_VEL
LIN {X 0,Y 105.378,Z 430.316,A -85,B 0,C 180,E1 -28108.916,E2 -28108.916} C_VEL
LIN {X 0,Y 104.824,Z 433.882,A -85,B 0,C 180,E1 -28111.963,E2 -28111.963} C_VEL
LIN {X 0,Y 100.859,Z 441.465,A -85,B 0,C 180,E1 -28116.741,E2 -28116.741} C_VEL
LIN {X 0,Y 98.839,Z 444.35,A -85,B 0,C 180,E1 -28118.54,E2 -28118.54} C_VEL
LIN {X 0,Y 91.753,Z 451.779,A -85,B 0,C 180,E1 -28123.31,E2 -28123.31} C_VEL
LIN {X 0,Y 85.395,Z 457.745,A -85,B 0,C 180,E1 -28128.82,E2 -28128.82} C_VEL
LIN {X 0,Y 79.779,Z 462.459,A -85,B 0,C 180,E1 -28135.066,E2 -28135.066} C_VEL
LIN {X 0,Y 75.226,Z 466.065,A -85,B 0,C 180,E1 -28142.15,E2 -28142.15} C_VEL
LIN {X 0,Y 72.967,Z 467.929,A -85,B 0,C 180,E1 -28147.337,E2 -28147.337} C_VEL
LIN {X 0,Y 70.207,Z 470.334,A -85,B 0,C 180,E1 -28158.449,E2 -28158.449} C_VEL
LIN {X 0,Y 69.655,Z 470.948,A -85,B 0,C 180,E1 -28164.207,E2 -28164.207} C_VEL
LIN {X 0,Y 69.7,Z 471.166,A -85,B 0,C 180,E1 -28169.997,E2 -28169.997} C_VEL
LIN {X 0,Y 69.654,Z 470.932,A -85,B 0,C 180,E1 -28175.788,E2 -28175.788} C_VEL
LIN {X 0,Y 70.206,Z 470.308,A -85,B 0,C 180,E1 -28181.547,E2 -28181.547} C_VEL
LIN {X 0,Y 71.284,Z 469.294,A -85,B 0,C 180,E1 -28187.201,E2 -28187.201} C_VEL
LIN {X 0,Y 72.965,Z 467.876,A -85,B 0,C 180,E1 -28192.658,E2 -28192.658} C_VEL
LIN {X 0,Y 76.622,Z 464.916,A -85,B 0,C 180,E1 -28200.293,E2 -28200.293} C_VEL
LIN {X 0,Y 81.493,Z 460.92,A -85,B 0,C 180,E1 -28207.13,E2 -28207.13} C_VEL
LIN {X 0,Y 87.44,Z 455.789,A -85,B 0,C 180,E1 -28213.09,E2 -28213.09} C_VEL
LIN {X 0,Y 93.982,Z 449.322,A -85,B 0,C 180,E1 -28218.397,E2 -28218.397} C_VEL
LIN {X 0,Y 99.919,Z 442.759,A -85,B 0,C 180,E1 -28222.302,E2 -28222.302} C_VEL
LIN {X 0,Y 103.564,Z 436.195,A -85,B 0,C 180,E1 -28226.505,E2 -28226.505} C_VEL
LIN {X 0,Y 104.743,Z 433.687,A -85,B 0,C 180,E1 -28228.033,E2 -28228.033} C_VEL
LIN {X 0,Y 105.326,Z 429.995,A -85,B 0,C 180,E1 -28231.156,E2 -28231.156} C_VEL
LIN {X 0,Y 105.614,Z 424.456,A -85,B 0,C 180,E1 -28236.468,E2 -28236.468} C_VEL
